DATA_BLOCK "_2015PU040U01_DB"   // DB4419
TITLE = Instance DB Unimotor:
{ S7_Optimized_Access := 'FALSE' }
AUTHOR : METIS
NAME : UNIMO_DB
VERSION : 8.0
// stored: InstanceOfName ACESYS_MOTOR
"ACESYS_MOTOR"
BEGIN
   FP_SEL.MD_OnOff := TRUE;
   FP_SEL.STW_Local := TRUE;
   FP_SEL.STW_Manual := TRUE;
   FP_SEL.STW_Single := TRUE;
   FP_SEL.Type_Unimotor := TRUE;
   FP_EN.Mode_Auto := TRUE;
   FP_EN.Mode_Man := TRUE;
   FP_EN.Mode_Loc := TRUE;
   FP_EN.Mode_SS_FP := TRUE;
   FP_SHOW.PB_Reset := TRUE;
   FP_PARM.StartWarn_Pre := 15;
   FP_PARM.RunDelay1_Pre := 5;
   FP_PARM.DelayStop_Pre := 5;
   FP_PARM.ReturnMon_Pre := 2;
   FP_PARM.AI1_Max := 19.8;
   FP_PARM.AI2_Max := 11.0;
   FP_PARM.AI3_Max := 2910.0;
   FP_PARM.AO1a_Max := 100.0;
   FP_PARM.AO2a_Max := 100.0;
   FP_PARM.AO3a_Max := 100.0;
   FP_PARM.AO1b_Max := 19.8;
   FP_PARM.AO2b_Max := 11.0;
   FP_PARM.AO3b_Max := 2910.0;
   MD := FALSE;
   SFS := FALSE;
   ES := TRUE;
   SPSET := 100.0;
   INTL.OK := TRUE;
   INTL_SEQ_STR1.OK := TRUE;
   INTL_SEQ_STR2.OK := TRUE;
   INTL_SEQ_STP.OK := TRUE;
   OK := TRUE;
   MAN := TRUE;
   CV := 100.0;
   MSW.EXT.ModeBit2 := TRUE;
   MSW.Status := 1;
   MSW.TimeStamp := 16#32F3;
   BlockInfo.Ace_Version := 80;
   BlockInfo.Ace_BuildNo := 13;
   BlockInfo.State_Act := 300;
   BlockInfo.State_Prev := 607;
   BlockInfo.DB_Number := 4419;
   FP_CMD.Manual := TRUE;
   FP_EN.PB_QStop := TRUE;
   FP_DIM.Auto := TRUE;
   FP_DIM.Local := TRUE;
   FP_DIM.Start1 := TRUE;
   FP_DIM.Start2 := TRUE;
   FP_DIM.Reset := TRUE;
   FP_SHOW.PB_Auto := TRUE;
   FP_SHOW.PB_Local := TRUE;
   FP_SHOW.PB_Manual := TRUE;
   FP_SHOW.PB_Start1 := TRUE;
   FP_SHOW.PB_Stop := TRUE;
   FP_SHOW.AI1 := TRUE;
   FP_SHOW.AI2 := TRUE;
   FP_SHOW.AI3 := TRUE;
   FP_SHOW.SP := TRUE;
   FP_SHOW.OVL := TRUE;
   FP_SHOW.SSW := TRUE;
   FP_SHOW.STALL := TRUE;
   FP_SHOW.EARTH := TRUE;
   FP_SHOW.UBAL := TRUE;
   FP_SHOW.GFA := TRUE;
   FP_SHOW.GWA := TRUE;
   FP_SHOW.BUSF := TRUE;
   FP_SHOW.DOPR := TRUE;
   FP_SHOW.DTEST := TRUE;
   FP_SHOW.LSTR1 := TRUE;
   FP_PARM.StartWarn_Acc := 15;
   FP_PARM.RunDelay1_Acc := 5;
   FP_PARM.DelayStop_Acc := 5;
   FP_PARM.ReturnMon_Acc := 2;
   FP_PARM.MD_Freq_SP := 1;
   FP_PARM.StopReason := 10;
   FP_PARM.INTL := TRUE;
   FP_PARM.INTL_SEQ_STR1 := TRUE;
   FP_PARM.INTL_SEQ_STR2 := TRUE;
   FP_PARM.INTL_SEQ_STP := TRUE;
   FP_SIM.OVL_Enable := TRUE;
   FP_SIM.RDY_Enable := TRUE;
   FP_SIM.SSW_Enable := TRUE;
   FP_SIM.TFA_Enable := TRUE;
   FP_SIM.MCC_Enable := TRUE;
   FP_SIM.DRDY_Enable := TRUE;
   FP_SIM.MD_Enable := TRUE;
   FP_SIM.GFA_Enable := TRUE;
   FP_SIM.GWA_Enable := TRUE;
   FP_SIM.STALL_Enable := TRUE;
   FP_SIM.EARTH_Enable := TRUE;
   FP_SIM.UBAL_Enable := TRUE;
   FP_SIM.BUSF_Enable := TRUE;
   FP_SIM.RET1_Enable := TRUE;
   FP_SIM.RET2_Enable := TRUE;
   FP_SIM.DOPR_Enable := TRUE;
   FP_SIM.ACK_Enable := TRUE;
   FP_SIM.LSTP_Enable := TRUE;
   FP_SIM.REM_Enable := TRUE;
   FP_SIM.SFS_Enable := TRUE;
   FP_SIM.SLS_Enable := TRUE;
   FP_SIM.ES_Enable := TRUE;
   FP_SIM.WORK.Flash_Slow := TRUE;
   AdapterBlock.Intell_Type := 282;
   AdapterBlock.VersionNo := 220;
   AdapterBlock.FuncType := 41;
   AdapterBlock.Options := 1;
   AdapterBlock.NetNo := 106;
   AdapterBlock.NodeNo := 16;
   AdapterBlock.Flash_Slow := TRUE;
   AdapterBlock.Flash_Fast := TRUE;
   AdapterBlock.MAN := TRUE;
   AdapterBlock.HMI_INT[4] := 2910;
   AdapterBlock.HMI_INT[5] := 687;
   AdapterBlock.HMI_INT[7] := 20000;
   AdapterBlock.HMI_REAL[8] := 2910.0;
   AdapterBlock.HMI_BOOL[1] := TRUE;
   AdapterBlock.HMI_BOOL[5] := TRUE;
   AdapterBlock.HMI_BOOL[6] := TRUE;
   AdapterBlock.HMI_BOOL[10] := TRUE;
   AdapterBlock.HMI_BOOL[13] := TRUE;
   AdapterBlock.HMI_BOOL[32] := TRUE;
   AdapterBlock.HMI_BOOL[34] := TRUE;
   AdapterBlock.HMI_BOOL[35] := TRUE;
   AdapterBlock.HMI_BOOL[37] := TRUE;
   AdapterBlock.HMI_BOOL[38] := TRUE;
   AdapterBlock.HMI_BOOL[39] := TRUE;
   AdapterBlock.HMI_BOOL[43] := TRUE;
   AdapterBlock.HMI_BOOL[65] := TRUE;
   AdapterBlock.HMI_BOOL[89] := TRUE;
   STATE.M_Stopped := TRUE;
   ONS.Unimotor := TRUE;
   ONS.MD_OnOff := TRUE;
   ONS.Cmd_Manual := TRUE;
   ONS.GLTP := TRUE;
   ONS.CMD_Start1 := TRUE;
   ONS.CMD_Start2 := TRUE;
   ONS.SecPulse1 := TRUE;
   StatusWork := 1;
   ModePointer := 52;
   StartWarn_Mem := 15;
   RunDelay1_Mem := 5;
   DelayStop_Mem := 5;
   ReturnMon_Mem := 2;
   ModeManual := TRUE;
   FromStateManual := TRUE;
   ChangeDir1_Done := TRUE;
   ChangeDir2_Done := TRUE;
   OUT.OK := TRUE;
   OUT.MAN := TRUE;
   OUT.INTL_OK_STAT := TRUE;
   OUT.INTL_SEQ_STR1_OK_STAT := TRUE;
   OUT.INTL_SEQ_STR2_OK_STAT := TRUE;
   OUT.INTL_SEQ_STP_OK_STAT := TRUE;
   MSW_Status_Trans := 1;
END_DATA_BLOCK

DATA_BLOCK "_2015PU041M01_DB"   // DB4420
TITLE = Instance DB Unimotor:
{ S7_Optimized_Access := 'FALSE' }
AUTHOR : METIS
NAME : UNIMO_DB
VERSION : 8.0
// stored: InstanceOfName ACESYS_MOTOR
"ACESYS_MOTOR"
BEGIN
   FP_SEL.MD_OnOff := TRUE;
   FP_SEL.STW_Local := TRUE;
   FP_SEL.STW_Manual := TRUE;
   FP_SEL.STW_Single := TRUE;
   FP_SEL.Type_Unimotor := TRUE;
   FP_EN.Mode_Auto := TRUE;
   FP_EN.Mode_Man := TRUE;
   FP_EN.Mode_Loc := TRUE;
   FP_EN.Mode_SS_FP := TRUE;
   FP_SHOW.PB_Reset := TRUE;
   FP_PARM.StartWarn_Pre := 15;
   FP_PARM.RunDelay1_Pre := 5;
   FP_PARM.DelayStop_Pre := 5;
   FP_PARM.ReturnMon_Pre := 2;
   FP_PARM.AI1_Max := 19.8;
   FP_PARM.AI2_Max := 11.0;
   FP_PARM.AI3_Max := 2910.0;
   FP_PARM.AO1a_Max := 100.0;
   FP_PARM.AO2a_Max := 100.0;
   FP_PARM.AO3a_Max := 100.0;
   FP_PARM.AO1b_Max := 19.8;
   FP_PARM.AO2b_Max := 11.0;
   FP_PARM.AO3b_Max := 2910.0;
   MD := FALSE;
   SFS := FALSE;
   ES := TRUE;
   SPSET := 100.0;
   INTL.OK := TRUE;
   INTL_SEQ_STR1.OK := TRUE;
   INTL_SEQ_STR2.OK := TRUE;
   INTL_SEQ_STP.OK := TRUE;
   OK := TRUE;
   MAN := TRUE;
   CV := 100.0;
   MSW.EXT.ModeBit2 := TRUE;
   MSW.Status := 1;
   MSW.TimeStamp := 16#32F3;
   BlockInfo.Ace_Version := 80;
   BlockInfo.Ace_BuildNo := 13;
   BlockInfo.State_Act := 300;
   BlockInfo.State_Prev := 607;
   BlockInfo.DB_Number := 4420;
   FP_CMD.Manual := TRUE;
   FP_EN.PB_QStop := TRUE;
   FP_DIM.Auto := TRUE;
   FP_DIM.Local := TRUE;
   FP_DIM.Start1 := TRUE;
   FP_DIM.Start2 := TRUE;
   FP_DIM.Reset := TRUE;
   FP_SHOW.PB_Auto := TRUE;
   FP_SHOW.PB_Local := TRUE;
   FP_SHOW.PB_Manual := TRUE;
   FP_SHOW.PB_Start1 := TRUE;
   FP_SHOW.PB_Stop := TRUE;
   FP_SHOW.AI1 := TRUE;
   FP_SHOW.AI2 := TRUE;
   FP_SHOW.AI3 := TRUE;
   FP_SHOW.SP := TRUE;
   FP_SHOW.OVL := TRUE;
   FP_SHOW.SSW := TRUE;
   FP_SHOW.STALL := TRUE;
   FP_SHOW.EARTH := TRUE;
   FP_SHOW.UBAL := TRUE;
   FP_SHOW.GFA := TRUE;
   FP_SHOW.GWA := TRUE;
   FP_SHOW.BUSF := TRUE;
   FP_SHOW.DOPR := TRUE;
   FP_SHOW.DTEST := TRUE;
   FP_SHOW.LSTR1 := TRUE;
   FP_PARM.StartWarn_Acc := 15;
   FP_PARM.RunDelay1_Acc := 5;
   FP_PARM.DelayStop_Acc := 5;
   FP_PARM.ReturnMon_Acc := 2;
   FP_PARM.MD_Freq_SP := 1;
   FP_PARM.StopReason := 11;
   FP_PARM.INTL := TRUE;
   FP_PARM.INTL_SEQ_STR1 := TRUE;
   FP_PARM.INTL_SEQ_STR2 := TRUE;
   FP_PARM.INTL_SEQ_STP := TRUE;
   FP_SIM.OVL_Enable := TRUE;
   FP_SIM.RDY_Enable := TRUE;
   FP_SIM.SSW_Enable := TRUE;
   FP_SIM.TFA_Enable := TRUE;
   FP_SIM.MCC_Enable := TRUE;
   FP_SIM.DRDY_Enable := TRUE;
   FP_SIM.MD_Enable := TRUE;
   FP_SIM.GFA_Enable := TRUE;
   FP_SIM.GWA_Enable := TRUE;
   FP_SIM.STALL_Enable := TRUE;
   FP_SIM.EARTH_Enable := TRUE;
   FP_SIM.UBAL_Enable := TRUE;
   FP_SIM.BUSF_Enable := TRUE;
   FP_SIM.RET1_Enable := TRUE;
   FP_SIM.RET2_Enable := TRUE;
   FP_SIM.DOPR_Enable := TRUE;
   FP_SIM.ACK_Enable := TRUE;
   FP_SIM.LSTP_Enable := TRUE;
   FP_SIM.REM_Enable := TRUE;
   FP_SIM.SFS_Enable := TRUE;
   FP_SIM.SLS_Enable := TRUE;
   FP_SIM.ES_Enable := TRUE;
   FP_SIM.WORK.Flash_Slow := TRUE;
   AdapterBlock.Intell_Type := 282;
   AdapterBlock.VersionNo := 220;
   AdapterBlock.FuncType := 41;
   AdapterBlock.Options := 1;
   AdapterBlock.NetNo := 106;
   AdapterBlock.NodeNo := 78;
   AdapterBlock.Flash_Slow := TRUE;
   AdapterBlock.Flash_Fast := TRUE;
   AdapterBlock.MAN := TRUE;
   AdapterBlock.HMI_INT[4] := 2910;
   AdapterBlock.HMI_INT[5] := 687;
   AdapterBlock.HMI_INT[7] := 20000;
   AdapterBlock.HMI_REAL[8] := 2910.0;
   AdapterBlock.HMI_REAL[9] := 100.0;
   AdapterBlock.HMI_REAL[10] := 100.0;
   AdapterBlock.HMI_BOOL[1] := TRUE;
   AdapterBlock.HMI_BOOL[5] := TRUE;
   AdapterBlock.HMI_BOOL[6] := TRUE;
   AdapterBlock.HMI_BOOL[10] := TRUE;
   AdapterBlock.HMI_BOOL[13] := TRUE;
   AdapterBlock.HMI_BOOL[32] := TRUE;
   AdapterBlock.HMI_BOOL[34] := TRUE;
   AdapterBlock.HMI_BOOL[35] := TRUE;
   AdapterBlock.HMI_BOOL[37] := TRUE;
   AdapterBlock.HMI_BOOL[38] := TRUE;
   AdapterBlock.HMI_BOOL[39] := TRUE;
   AdapterBlock.HMI_BOOL[43] := TRUE;
   AdapterBlock.HMI_BOOL[65] := TRUE;
   AdapterBlock.HMI_BOOL[89] := TRUE;
   STATE.M_Stopped := TRUE;
   ONS.Unimotor := TRUE;
   ONS.MD_OnOff := TRUE;
   ONS.Cmd_Manual := TRUE;
   ONS.GLTP := TRUE;
   ONS.CMD_Start1 := TRUE;
   ONS.CMD_Start2 := TRUE;
   ONS.SecPulse1 := TRUE;
   StatusWork := 1;
   ModePointer := 52;
   StartWarn_Mem := 15;
   RunDelay1_Mem := 5;
   DelayStop_Mem := 5;
   ReturnMon_Mem := 2;
   ModeManual := TRUE;
   FromStateManual := TRUE;
   ChangeDir1_Done := TRUE;
   ChangeDir2_Done := TRUE;
   OUT.OK := TRUE;
   OUT.MAN := TRUE;
   OUT.INTL_OK_STAT := TRUE;
   OUT.INTL_SEQ_STR1_OK_STAT := TRUE;
   OUT.INTL_SEQ_STR2_OK_STAT := TRUE;
   OUT.INTL_SEQ_STP_OK_STAT := TRUE;
   MSW_Status_Trans := 1;
END_DATA_BLOCK

DATA_BLOCK "_2015PU042M01_DB"   // DB4421
TITLE = Instance DB Unimotor:
{ S7_Optimized_Access := 'FALSE' }
AUTHOR : METIS
NAME : UNIMO_DB
VERSION : 8.0
// stored: InstanceOfName ACESYS_MOTOR
"ACESYS_MOTOR"
BEGIN
   FP_SEL.MD_OnOff := TRUE;
   FP_SEL.STW_Local := TRUE;
   FP_SEL.STW_Manual := TRUE;
   FP_SEL.STW_Single := TRUE;
   FP_SEL.Type_Unimotor := TRUE;
   FP_EN.Mode_Auto := TRUE;
   FP_EN.Mode_Man := TRUE;
   FP_EN.Mode_Loc := TRUE;
   FP_EN.Mode_SS_FP := TRUE;
   FP_SHOW.PB_Reset := TRUE;
   FP_PARM.StartWarn_Pre := 15;
   FP_PARM.RunDelay1_Pre := 5;
   FP_PARM.DelayStop_Pre := 5;
   FP_PARM.ReturnMon_Pre := 2;
   FP_PARM.AI1_Max := 100.0;
   FP_PARM.AI2_Max := 100.0;
   FP_PARM.AI3_Max := 100.0;
   FP_PARM.AO1a_Max := 100.0;
   FP_PARM.AO2a_Max := 100.0;
   FP_PARM.AO3a_Max := 100.0;
   FP_PARM.AO1b_Max := 100.0;
   FP_PARM.AO2b_Max := 100.0;
   FP_PARM.AO3b_Max := 100.0;
   MD := FALSE;
   SFS := FALSE;
   ES := TRUE;
   INTL.OK := TRUE;
   INTL_SEQ_STR1.OK := TRUE;
   INTL_SEQ_STR2.OK := TRUE;
   INTL_SEQ_STP.OK := TRUE;
   OK := TRUE;
   MAN := TRUE;
   MSW.EXT.ModeBit2 := TRUE;
   MSW.Status := 1;
   MSW.TimeStamp := 16#9BB1;
   BlockInfo.Ace_Version := 80;
   BlockInfo.Ace_BuildNo := 13;
   BlockInfo.State_Act := 300;
   BlockInfo.State_Prev := 607;
   BlockInfo.DB_Number := 4421;
   FP_CMD.Manual := TRUE;
   FP_EN.PB_QStop := TRUE;
   FP_DIM.Auto := TRUE;
   FP_DIM.Local := TRUE;
   FP_DIM.Start1 := TRUE;
   FP_DIM.Start2 := TRUE;
   FP_DIM.Reset := TRUE;
   FP_SHOW.PB_Auto := TRUE;
   FP_SHOW.PB_Local := TRUE;
   FP_SHOW.PB_Manual := TRUE;
   FP_SHOW.PB_Start1 := TRUE;
   FP_SHOW.PB_Stop := TRUE;
   FP_SHOW.OVL := TRUE;
   FP_SHOW.LSTP := TRUE;
   FP_SHOW.SSW := TRUE;
   FP_SHOW.DRDY := TRUE;
   FP_SHOW.STALL := TRUE;
   FP_SHOW.EARTH := TRUE;
   FP_SHOW.UBAL := TRUE;
   FP_SHOW.GFA := TRUE;
   FP_SHOW.GWA := TRUE;
   FP_SHOW.BUSF := TRUE;
   FP_SHOW.DOPR := TRUE;
   FP_SHOW.DTEST := TRUE;
   FP_SHOW.LSTR1 := TRUE;
   FP_PARM.StartWarn_Acc := 15;
   FP_PARM.RunDelay1_Acc := 5;
   FP_PARM.DelayStop_Acc := 5;
   FP_PARM.ReturnMon_Acc := 2;
   FP_PARM.MD_Freq_SP := 1;
   FP_PARM.StopReason := 99;
   FP_PARM.INTL := TRUE;
   FP_PARM.INTL_SEQ_STR1 := TRUE;
   FP_PARM.INTL_SEQ_STR2 := TRUE;
   FP_PARM.INTL_SEQ_STP := TRUE;
   FP_SIM.OVL_Enable := TRUE;
   FP_SIM.RDY_Enable := TRUE;
   FP_SIM.SSW_Enable := TRUE;
   FP_SIM.TFA_Enable := TRUE;
   FP_SIM.MCC_Enable := TRUE;
   FP_SIM.DRDY_Enable := TRUE;
   FP_SIM.MD_Enable := TRUE;
   FP_SIM.GFA_Enable := TRUE;
   FP_SIM.GWA_Enable := TRUE;
   FP_SIM.STALL_Enable := TRUE;
   FP_SIM.EARTH_Enable := TRUE;
   FP_SIM.UBAL_Enable := TRUE;
   FP_SIM.BUSF_Enable := TRUE;
   FP_SIM.RET1_Enable := TRUE;
   FP_SIM.RET2_Enable := TRUE;
   FP_SIM.DOPR_Enable := TRUE;
   FP_SIM.ACK_Enable := TRUE;
   FP_SIM.LSTP_Enable := TRUE;
   FP_SIM.REM_Enable := TRUE;
   FP_SIM.SFS_Enable := TRUE;
   FP_SIM.SLS_Enable := TRUE;
   FP_SIM.ES_Enable := TRUE;
   AdapterBlock.Intell_Type := 54;
   AdapterBlock.VersionNo := 420;
   AdapterBlock.BuildNo := 1;
   AdapterBlock.FuncType := 41;
   AdapterBlock.NetNo := 106;
   AdapterBlock.NodeNo := 64;
   AdapterBlock.MAN := TRUE;
   AdapterBlock.HMI_BOOL[4] := TRUE;
   AdapterBlock.HMI_BOOL[8] := TRUE;
   AdapterBlock.HMI_BOOL[18] := TRUE;
   AdapterBlock.HMI_BOOL[19] := TRUE;
   AdapterBlock.HMI_BOOL[20] := TRUE;
   AdapterBlock.HMI_BOOL[28] := TRUE;
   AdapterBlock.HMI_BOOL[74] := TRUE;
   STATE.M_Stopped := TRUE;
   ONS.Unimotor := TRUE;
   ONS.MD_OnOff := TRUE;
   ONS.Cmd_Manual := TRUE;
   ONS.GLTP := TRUE;
   ONS.CMD_Start1 := TRUE;
   ONS.CMD_Start2 := TRUE;
   ONS.SecPulse1 := TRUE;
   StatusWork := 1;
   ModePointer := 52;
   StartWarn_Mem := 15;
   RunDelay1_Mem := 5;
   DelayStop_Mem := 5;
   ReturnMon_Mem := 2;
   ModeManual := TRUE;
   FromStateManual := TRUE;
   ChangeDir1_Done := TRUE;
   ChangeDir2_Done := TRUE;
   OUT.OK := TRUE;
   OUT.MAN := TRUE;
   OUT.INTL_OK_STAT := TRUE;
   OUT.INTL_SEQ_STR1_OK_STAT := TRUE;
   OUT.INTL_SEQ_STR2_OK_STAT := TRUE;
   OUT.INTL_SEQ_STP_OK_STAT := TRUE;
   MSW_Status_Trans := 1;
END_DATA_BLOCK

DATA_BLOCK "_MTR_SPARE_DB"   // DB4422
TITLE = Instance DB Unimotor:
{ S7_Optimized_Access := 'FALSE' }
AUTHOR : METIS
NAME : UNIMO_DB
VERSION : 8.0
// stored: InstanceOfName ACESYS_MOTOR
"ACESYS_MOTOR"
BEGIN
   FP_SEL.MD_OnOff := TRUE;
   FP_SEL.STW_Local := TRUE;
   FP_SEL.STW_Manual := TRUE;
   FP_SEL.STW_Single := TRUE;
   FP_SEL.Type_Unimotor := TRUE;
   FP_EN.Mode_Auto := TRUE;
   FP_EN.Mode_Man := TRUE;
   FP_EN.Mode_Loc := TRUE;
   FP_EN.Mode_SS_FP := TRUE;
   FP_SHOW.PB_Reset := TRUE;
   FP_PARM.StartWarn_Pre := 15;
   FP_PARM.RunDelay1_Pre := 5;
   FP_PARM.DelayStop_Pre := 5;
   FP_PARM.ReturnMon_Pre := 2;
   FP_PARM.AI1_Max := 100.0;
   FP_PARM.AI2_Max := 100.0;
   FP_PARM.AI3_Max := 100.0;
   FP_PARM.AO1a_Max := 100.0;
   FP_PARM.AO2a_Max := 100.0;
   FP_PARM.AO3a_Max := 100.0;
   FP_PARM.AO1b_Max := 100.0;
   FP_PARM.AO2b_Max := 100.0;
   FP_PARM.AO3b_Max := 100.0;
   MD := FALSE;
   SFS := FALSE;
   ES := TRUE;
   INTL.OK := TRUE;
   INTL_SEQ_STR1.OK := TRUE;
   INTL_SEQ_STR2.OK := TRUE;
   INTL_SEQ_STP.OK := TRUE;
   OK := TRUE;
   MAN := TRUE;
   MSW.EXT.ModeBit2 := TRUE;
   MSW.Status := 1;
   MSW.TimeStamp := 16#9BB1;
   BlockInfo.Ace_Version := 80;
   BlockInfo.Ace_BuildNo := 13;
   BlockInfo.State_Act := 300;
   BlockInfo.State_Prev := 607;
   BlockInfo.DB_Number := 4421;
   FP_CMD.Manual := TRUE;
   FP_EN.PB_QStop := TRUE;
   FP_DIM.Auto := TRUE;
   FP_DIM.Local := TRUE;
   FP_DIM.Start1 := TRUE;
   FP_DIM.Start2 := TRUE;
   FP_DIM.Reset := TRUE;
   FP_SHOW.PB_Auto := TRUE;
   FP_SHOW.PB_Local := TRUE;
   FP_SHOW.PB_Manual := TRUE;
   FP_SHOW.PB_Start1 := TRUE;
   FP_SHOW.PB_Stop := TRUE;
   FP_SHOW.OVL := TRUE;
   FP_SHOW.LSTP := TRUE;
   FP_SHOW.SSW := TRUE;
   FP_SHOW.DRDY := TRUE;
   FP_SHOW.STALL := TRUE;
   FP_SHOW.EARTH := TRUE;
   FP_SHOW.UBAL := TRUE;
   FP_SHOW.GFA := TRUE;
   FP_SHOW.GWA := TRUE;
   FP_SHOW.BUSF := TRUE;
   FP_SHOW.DOPR := TRUE;
   FP_SHOW.DTEST := TRUE;
   FP_SHOW.LSTR1 := TRUE;
   FP_PARM.StartWarn_Acc := 15;
   FP_PARM.RunDelay1_Acc := 5;
   FP_PARM.DelayStop_Acc := 5;
   FP_PARM.ReturnMon_Acc := 2;
   FP_PARM.MD_Freq_SP := 1;
   FP_PARM.StopReason := 99;
   FP_PARM.INTL := TRUE;
   FP_PARM.INTL_SEQ_STR1 := TRUE;
   FP_PARM.INTL_SEQ_STR2 := TRUE;
   FP_PARM.INTL_SEQ_STP := TRUE;
   FP_SIM.OVL_Enable := TRUE;
   FP_SIM.RDY_Enable := TRUE;
   FP_SIM.SSW_Enable := TRUE;
   FP_SIM.TFA_Enable := TRUE;
   FP_SIM.MCC_Enable := TRUE;
   FP_SIM.DRDY_Enable := TRUE;
   FP_SIM.MD_Enable := TRUE;
   FP_SIM.GFA_Enable := TRUE;
   FP_SIM.GWA_Enable := TRUE;
   FP_SIM.STALL_Enable := TRUE;
   FP_SIM.EARTH_Enable := TRUE;
   FP_SIM.UBAL_Enable := TRUE;
   FP_SIM.BUSF_Enable := TRUE;
   FP_SIM.RET1_Enable := TRUE;
   FP_SIM.RET2_Enable := TRUE;
   FP_SIM.DOPR_Enable := TRUE;
   FP_SIM.ACK_Enable := TRUE;
   FP_SIM.LSTP_Enable := TRUE;
   FP_SIM.REM_Enable := TRUE;
   FP_SIM.SFS_Enable := TRUE;
   FP_SIM.SLS_Enable := TRUE;
   FP_SIM.ES_Enable := TRUE;
   AdapterBlock.Intell_Type := 54;
   AdapterBlock.VersionNo := 420;
   AdapterBlock.BuildNo := 1;
   AdapterBlock.FuncType := 41;
   AdapterBlock.NetNo := 106;
   AdapterBlock.NodeNo := 64;
   AdapterBlock.MAN := TRUE;
   AdapterBlock.HMI_BOOL[4] := TRUE;
   AdapterBlock.HMI_BOOL[8] := TRUE;
   AdapterBlock.HMI_BOOL[18] := TRUE;
   AdapterBlock.HMI_BOOL[19] := TRUE;
   AdapterBlock.HMI_BOOL[20] := TRUE;
   AdapterBlock.HMI_BOOL[28] := TRUE;
   AdapterBlock.HMI_BOOL[74] := TRUE;
   STATE.M_Stopped := TRUE;
   ONS.Unimotor := TRUE;
   ONS.MD_OnOff := TRUE;
   ONS.Cmd_Manual := TRUE;
   ONS.GLTP := TRUE;
   ONS.CMD_Start1 := TRUE;
   ONS.CMD_Start2 := TRUE;
   ONS.SecPulse1 := TRUE;
   StatusWork := 1;
   ModePointer := 52;
   StartWarn_Mem := 15;
   RunDelay1_Mem := 5;
   DelayStop_Mem := 5;
   ReturnMon_Mem := 2;
   ModeManual := TRUE;
   FromStateManual := TRUE;
   ChangeDir1_Done := TRUE;
   ChangeDir2_Done := TRUE;
   OUT.OK := TRUE;
   OUT.MAN := TRUE;
   OUT.INTL_OK_STAT := TRUE;
   OUT.INTL_SEQ_STR1_OK_STAT := TRUE;
   OUT.INTL_SEQ_STR2_OK_STAT := TRUE;
   OUT.INTL_SEQ_STP_OK_STAT := TRUE;
   MSW_Status_Trans := 1;
END_DATA_BLOCK

DATA_BLOCK "_2015PU035U01_DB"   // DB4433
TITLE = Instance DB Unimotor:
{ S7_Optimized_Access := 'FALSE' }
AUTHOR : METIS
NAME : UNIMO_DB
VERSION : 8.0
// stored: InstanceOfName ACESYS_MOTOR
"ACESYS_MOTOR"
BEGIN
   FP_SEL.MD_OnOff := TRUE;
   FP_SEL.STW_Local := TRUE;
   FP_SEL.STW_Manual := TRUE;
   FP_SEL.STW_Single := TRUE;
   FP_SEL.Type_Unimotor := TRUE;
   FP_EN.Mode_Auto := TRUE;
   FP_EN.Mode_Man := TRUE;
   FP_EN.Mode_Loc := TRUE;
   FP_EN.Mode_SS_FP := TRUE;
   FP_SHOW.PB_Reset := TRUE;
   FP_PARM.StartWarn_Pre := 15;
   FP_PARM.RunDelay1_Pre := 5;
   FP_PARM.DelayStop_Pre := 5;
   FP_PARM.ReturnMon_Pre := 2;
   FP_PARM.AI1_Max := 100.0;
   FP_PARM.AI2_Max := 100.0;
   FP_PARM.AI3_Max := 100.0;
   FP_PARM.AO1a_Max := 100.0;
   FP_PARM.AO2a_Max := 100.0;
   FP_PARM.AO3a_Max := 100.0;
   FP_PARM.AO1b_Max := 100.0;
   FP_PARM.AO2b_Max := 100.0;
   FP_PARM.AO3b_Max := 100.0;
   MD := FALSE;
   SFS := FALSE;
   SLS := TRUE;
   ES := TRUE;
   SPSET := 20.0;
   INTL.OK := TRUE;
   INTL_SEQ_STR1.OK := TRUE;
   INTL_SEQ_STR2.OK := TRUE;
   INTL_SEQ_STP.OK := TRUE;
   OK := TRUE;
   MAN := TRUE;
   CV := 20.0;
   MSW.EXT.ModeBit2 := TRUE;
   MSW.Status := 1;
   MSW.TimeStamp := 16#A9DD;
   BlockInfo.Ace_Version := 80;
   BlockInfo.Ace_BuildNo := 13;
   BlockInfo.State_Act := 300;
   BlockInfo.State_Prev := 305;
   BlockInfo.DB_Number := 4433;
   FP_CMD.Manual := TRUE;
   FP_EN.PB_QStop := TRUE;
   FP_DIM.Auto := TRUE;
   FP_DIM.Local := TRUE;
   FP_DIM.Start1 := TRUE;
   FP_DIM.Start2 := TRUE;
   FP_DIM.Reset := TRUE;
   FP_SHOW.PB_Auto := TRUE;
   FP_SHOW.PB_Local := TRUE;
   FP_SHOW.PB_Manual := TRUE;
   FP_SHOW.PB_Start1 := TRUE;
   FP_SHOW.PB_Stop := TRUE;
   FP_SHOW.AI1 := TRUE;
   FP_SHOW.AI2 := TRUE;
   FP_SHOW.AI3 := TRUE;
   FP_SHOW.SP := TRUE;
   FP_SHOW.OVL := TRUE;
   FP_SHOW.SSW := TRUE;
   FP_SHOW.STALL := TRUE;
   FP_SHOW.EARTH := TRUE;
   FP_SHOW.UBAL := TRUE;
   FP_SHOW.GFA := TRUE;
   FP_SHOW.GWA := TRUE;
   FP_SHOW.BUSF := TRUE;
   FP_SHOW.DOPR := TRUE;
   FP_SHOW.DTEST := TRUE;
   FP_SHOW.LSTR1 := TRUE;
   FP_PARM.StartWarn_Acc := 15;
   FP_PARM.RunDelay1_Acc := 5;
   FP_PARM.DelayStop_Acc := 5;
   FP_PARM.ReturnMon_Acc := 2;
   FP_PARM.MD_Freq_SP := 1;
   FP_PARM.StopReason := 3;
   FP_PARM.INTL := TRUE;
   FP_PARM.INTL_SEQ_STR1 := TRUE;
   FP_PARM.INTL_SEQ_STR2 := TRUE;
   FP_PARM.INTL_SEQ_STP := TRUE;
   FP_SIM.OVL_Enable := TRUE;
   FP_SIM.RDY_Enable := TRUE;
   FP_SIM.SSW_Enable := TRUE;
   FP_SIM.TFA_Enable := TRUE;
   FP_SIM.MCC_Enable := TRUE;
   FP_SIM.DRDY_Enable := TRUE;
   FP_SIM.MD_Enable := TRUE;
   FP_SIM.GFA_Enable := TRUE;
   FP_SIM.GWA_Enable := TRUE;
   FP_SIM.STALL_Enable := TRUE;
   FP_SIM.EARTH_Enable := TRUE;
   FP_SIM.UBAL_Enable := TRUE;
   FP_SIM.BUSF_Enable := TRUE;
   FP_SIM.RET1_Enable := TRUE;
   FP_SIM.RET2_Enable := TRUE;
   FP_SIM.DOPR_Enable := TRUE;
   FP_SIM.ACK_Enable := TRUE;
   FP_SIM.LSTP_Enable := TRUE;
   FP_SIM.REM_Enable := TRUE;
   FP_SIM.SFS_Enable := TRUE;
   FP_SIM.SLS_Enable := TRUE;
   FP_SIM.ES_Enable := TRUE;
   AdapterBlock.Intell_Type := 282;
   AdapterBlock.VersionNo := 220;
   AdapterBlock.FuncType := 41;
   AdapterBlock.Options := 1;
   AdapterBlock.NetNo := 106;
   AdapterBlock.NodeNo := 75;
   AdapterBlock.MAN := TRUE;
   AdapterBlock.HMI_INT[7] := 1000;
   AdapterBlock.HMI_INT[9] := 3;
   AdapterBlock.HMI_INT[10] := 2;
   AdapterBlock.HMI_INT[11] := 6;
   AdapterBlock.HMI_REAL[9] := 100.0;
   AdapterBlock.HMI_REAL[10] := 100.0;
   AdapterBlock.HMI_REAL[12] := 100.0;
   AdapterBlock.HMI_BOOL[1] := TRUE;
   AdapterBlock.HMI_BOOL[2] := TRUE;
   AdapterBlock.HMI_BOOL[9] := TRUE;
   AdapterBlock.HMI_BOOL[15] := TRUE;
   AdapterBlock.HMI_BOOL[17] := TRUE;
   AdapterBlock.HMI_BOOL[18] := TRUE;
   AdapterBlock.HMI_BOOL[34] := TRUE;
   AdapterBlock.HMI_BOOL[35] := TRUE;
   AdapterBlock.HMI_BOOL[65] := TRUE;
   AdapterBlock.HMI_BOOL[89] := TRUE;
   STATE.M_Stopped := TRUE;
   ONS.Unimotor := TRUE;
   ONS.MD_OnOff := TRUE;
   ONS.Cmd_Manual := TRUE;
   ONS.GLTP := TRUE;
   ONS.CMD_Start1 := TRUE;
   ONS.CMD_Start2 := TRUE;
   ONS.SecPulse1 := TRUE;
   StatusWork := 1;
   ModePointer := 52;
   StartWarn_Mem := 15;
   RunDelay1_Mem := 5;
   DelayStop_Mem := 5;
   ReturnMon_Mem := 2;
   ModeManual := TRUE;
   FromStateManual := TRUE;
   ChangeDir1_Done := TRUE;
   ChangeDir2_Done := TRUE;
   OUT.OK := TRUE;
   OUT.MAN := TRUE;
   OUT.INTL_OK_STAT := TRUE;
   OUT.INTL_SEQ_STR1_OK_STAT := TRUE;
   OUT.INTL_SEQ_STR2_OK_STAT := TRUE;
   OUT.INTL_SEQ_STP_OK_STAT := TRUE;
   MSW_Status_Trans := 1;
END_DATA_BLOCK

DATA_BLOCK "_2015PU027Y01_DB"   // DB4434
{ S7_Optimized_Access := 'FALSE' }
AUTHOR : FLSmidth
FAMILY : ACESYS
NAME : VALVE
VERSION : 8.0
// stored: InstanceOfName ACESYS_VALVE
"ACESYS_VALVE"
BEGIN
END_DATA_BLOCK

DATA_BLOCK "_2015PU028Y01_DB"   // DB4435
{ S7_Optimized_Access := 'FALSE' }
AUTHOR : FLSmidth
FAMILY : ACESYS
NAME : VALVE
VERSION : 8.0
// stored: InstanceOfName ACESYS_VALVE
"ACESYS_VALVE"
BEGIN
END_DATA_BLOCK

DATA_BLOCK "_2010CV300N01T01_DB"   // DB5000
TITLE = Instance DB Analog:
{ S7_Optimized_Access := 'FALSE' }
AUTHOR : METIS
NAME : ANA_DB
VERSION : 8.0
// stored: InstanceOfName ACESYS_ANALOG
"ACESYS_ANALOG"
BEGIN
   FP_EN.ParentSupress := TRUE;
   FP_EN.ParentSupressUnit := TRUE;
   FP_EN.Hysteresis := TRUE;
   FP_PARM.Scale_Max := 200.0;
   FP_PARM.Grad_Pos := 0.0;
   FP_PARM.Grad_Neg := 0.0;
   FP_PARM.OpenLoopDelay_Pre := 2;
   FP_PARM.Gradient_Time_Pre := 10;
   FP_PARM.Alarm_Hyst := 1.0;
   FP_PARM.OverRangeDelay_Pre := 2;
   FP_SIM.Value_Enable := TRUE;
   FP_SIM.Gain := 1.0;
   IN := 41.90176;
   U_RANGE := TRUE;
   O_RANGE := TRUE;
   SIG_FAULT := TRUE;
   EnConfig := TRUE;
   AEN := TRUE;
   PV_NORM := 41.90176;
   PV_SCAL := 54.75442;
   AL_H3 := TRUE;
   AL_H2 := TRUE;
   AL_H1 := TRUE;
   AL_L1 := TRUE;
   AL_L2 := TRUE;
   AL_L3 := TRUE;
   SIG_OK := TRUE;
   LIM_H2 := TRUE;
   LIM_H1 := TRUE;
   MSW.VALUE := 54.75442;
   MSW.TRIGVALUE := -53.03819;
   MSW.EXT.AlarmWarnUnAck := TRUE;
   MSW.EXT.Operation := TRUE;
   MSW.Status := 1;
   MSW.TimeStamp := 16#97DF;
   BlockInfo.Ace_Version := 80;
   BlockInfo.Ace_BuildNo := 3;
   BlockInfo.DB_Number := 5000;
   FP_EN.Alarm_H2 := TRUE;
   FP_EN.Alarm_H1 := TRUE;
   FP_EN.AlarmDelay_H2 := TRUE;
   FP_EN.AlarmDelay_H1 := TRUE;
   FP_PARM.Scale_Min := -50.0;
   FP_PARM.Gradient_Time_ACC := 10;
   FP_PARM.AlarmLimit_H2 := 85.0;
   FP_PARM.AlarmLimit_H1 := 80.0;
   FP_PARM.AlarmDelay_H2_Pre := 2;
   FP_PARM.AlarmDelay_H2_Acc := 2;
   FP_PARM.AlarmDelay_H1_Pre := 2;
   FP_PARM.AlarmDelay_H1_Acc := 2;
   FP_PARM.OpenLoopDelay_Acc := 2;
   FP_PARM.OverRangeDelay_Acc := 2;
   ONS.SecPulse1 := TRUE;
   FIBUS_SubStatus := 16#FF;
   FIBUS_Quality := 16#FF;
   FIBUS_Limit := 16#FF;
   Result_Smooth := 41.90176;
   DampXEA := 41.90176;
   StatusWork := 1;
   AlarmDelay_H2_Mem := 2;
   AlarmDelay_H1_Mem := 2;
   GradientTime_Mem := 10;
   AlarmDelay_OpenLoop_Mem := 2;
   AlarmDelay_OverRange_Mem := 2;
   ScaledValue := 54.75442;
   Grad_OldValue := 54.75442;
   HystCalc := 2.5;
   OUT.PV_NORM := 41.90176;
   OUT.PV_SCAL := 54.75442;
   OUT.AL_H3 := TRUE;
   OUT.AL_H2 := TRUE;
   OUT.AL_H1 := TRUE;
   OUT.AL_L1 := TRUE;
   OUT.AL_L2 := TRUE;
   OUT.AL_L3 := TRUE;
   OUT.SIG_OK := TRUE;
   OUT.LIM_H2 := TRUE;
   OUT.LIM_H1 := TRUE;
   MSW_Status_Trans := 1;
END_DATA_BLOCK

DATA_BLOCK "_2010CV300U01I01_DB"   // DB5001
TITLE = Instance DB Analog:
{ S7_Optimized_Access := 'FALSE' }
AUTHOR : METIS
NAME : ANA_DB
VERSION : 8.0
// stored: InstanceOfName ACESYS_ANALOG
"ACESYS_ANALOG"
BEGIN
   FP_EN.Hysteresis := TRUE;
   FP_PARM.Scale_Max := 487.0;
   FP_PARM.Grad_Pos := 0.0;
   FP_PARM.Grad_Neg := 0.0;
   FP_PARM.OpenLoopDelay_Pre := 2;
   FP_PARM.Gradient_Time_Pre := 10;
   FP_PARM.Alarm_Hyst := 1.0;
   FP_PARM.OverRangeDelay_Pre := 2;
   FP_SIM.Value_Enable := TRUE;
   FP_SIM.Gain := 1.0;
   SIG_TYPE := 1;
   IN := 251.3;
   U_RANGE := TRUE;
   O_RANGE := TRUE;
   SIG_FAULT := TRUE;
   EnConfig := TRUE;
   AEN := TRUE;
   PV_NORM := 51.60164;
   PV_SCAL := 251.3;
   AL_H3 := TRUE;
   AL_H2 := TRUE;
   AL_H1 := TRUE;
   AL_L1 := TRUE;
   AL_L2 := TRUE;
   AL_L3 := TRUE;
   SIG_OK := TRUE;
   LIM_H2 := TRUE;
   LIM_H1 := TRUE;
   MSW.VALUE := 251.3;
   MSW.TRIGVALUE := 294.1;
   MSW.EXT.AlarmWarnUnAck := TRUE;
   MSW.EXT.Operation := TRUE;
   MSW.Status := 1;
   MSW.TimeStamp := 16#ADFA;
   BlockInfo.Ace_Version := 80;
   BlockInfo.Ace_BuildNo := 3;
   BlockInfo.DB_Number := 5001;
   FP_EN.Alarm_H3 := TRUE;
   FP_EN.Alarm_H2 := TRUE;
   FP_EN.Alarm_H1 := TRUE;
   FP_EN.AlarmDelay_H3 := TRUE;
   FP_EN.AlarmDelay_H2 := TRUE;
   FP_EN.U_Range_Warn := FALSE;
   FP_EN.O_Range_Warn := FALSE;
   FP_PARM.Gradient_Time_ACC := 10;
   FP_PARM.AlarmLimit_H3 := 350.0;
   FP_PARM.AlarmLimit_H2 := 320.0;
   FP_PARM.AlarmLimit_H1 := 300.0;
   FP_PARM.AlarmDelay_H3_Pre := 30;
   FP_PARM.AlarmDelay_H3_Acc := 30;
   FP_PARM.AlarmDelay_H2_Pre := 1;
   FP_PARM.AlarmDelay_H2_Acc := 1;
   FP_PARM.OpenLoopDelay_Acc := 2;
   FP_PARM.OverRangeDelay_Acc := 2;
   ONS.SecPulse1 := TRUE;
   FIBUS_SubStatus := 16#FF;
   FIBUS_Quality := 16#FF;
   FIBUS_Limit := 16#FF;
   Result_Smooth := 51.60164;
   DampXEA := 51.60164;
   StatusWork := 1;
   AlarmDelay_H3_Mem := 30;
   AlarmDelay_H2_Mem := 1;
   GradientTime_Mem := 10;
   AlarmDelay_OpenLoop_Mem := 2;
   AlarmDelay_OverRange_Mem := 2;
   ScaledValue := 251.3;
   Grad_OldValue := 251.3;
   HystCalc := 4.87;
   OUT.PV_NORM := 51.60164;
   OUT.PV_SCAL := 251.3;
   OUT.AL_H3 := TRUE;
   OUT.AL_H2 := TRUE;
   OUT.AL_H1 := TRUE;
   OUT.AL_L1 := TRUE;
   OUT.AL_L2 := TRUE;
   OUT.AL_L3 := TRUE;
   OUT.SIG_OK := TRUE;
   OUT.LIM_H2 := TRUE;
   OUT.LIM_H1 := TRUE;
   MSW_Status_Trans := 1;
END_DATA_BLOCK

DATA_BLOCK "_2010CV300U01J01_DB"   // DB5002
TITLE = Instance DB Analog:
{ S7_Optimized_Access := 'FALSE' }
AUTHOR : METIS
NAME : ANA_DB
VERSION : 8.0
// stored: InstanceOfName ACESYS_ANALOG
"ACESYS_ANALOG"
BEGIN
   FP_EN.ParentSupress := TRUE;
   FP_EN.ParentSupressUnit := TRUE;
   FP_EN.Hysteresis := TRUE;
   FP_PARM.OverRangeDelay_Pre := 2;
   FP_PARM.Grad_Pos := 0.0;
   FP_PARM.Grad_Neg := 0.0;
   FP_PARM.OpenLoopDelay_Pre := 2;
   FP_PARM.Gradient_Time_Pre := 10;
   FP_PARM.Alarm_Hyst := 1.0;
   FP_SIM.Value_Enable := TRUE;
   FP_SIM.Gain := 1.0;
   SIG_TYPE := 1;
   IN := 140.0;
   U_RANGE := TRUE;
   O_RANGE := TRUE;
   SIG_FAULT := TRUE;
   EnConfig := TRUE;
   AEN := TRUE;
   PV_NORM := 140.0;
   PV_SCAL := 140.0;
   AL_H3 := TRUE;
   AL_H2 := TRUE;
   AL_H1 := TRUE;
   AL_L1 := TRUE;
   AL_L2 := TRUE;
   AL_L3 := TRUE;
   SIG_OK := TRUE;
   LIM_H2 := TRUE;
   LIM_H1 := TRUE;
   MSW.VALUE := 140.0;
   MSW.EXT.AlarmWarnUnAck := TRUE;
   MSW.EXT.Operation := TRUE;
   MSW.Status := 1;
   MSW.TimeStamp := 16#3928;
   BlockInfo.Ace_Version := 80;
   BlockInfo.Ace_BuildNo := 3;
   BlockInfo.DB_Number := 5002;
   FP_EN.U_Range_Warn := FALSE;
   FP_EN.O_Range_Warn := FALSE;
   FP_PARM.Gradient_Time_ACC := 10;
   FP_PARM.OpenLoopDelay_Acc := 2;
   FP_PARM.OverRangeDelay_Acc := 2;
   ONS.SecPulse1 := TRUE;
   FIBUS_SubStatus := 16#FF;
   FIBUS_Quality := 16#FF;
   FIBUS_Limit := 16#FF;
   Result_Smooth := 140.0;
   DampXEA := 140.0;
   StatusWork := 1;
   GradientTime_Mem := 10;
   AlarmDelay_OpenLoop_Mem := 2;
   AlarmDelay_OverRange_Mem := 2;
   ScaledValue := 140.0;
   Grad_OldValue := 140.0;
   HystCalc := 1.0;
   OUT.PV_NORM := 140.0;
   OUT.PV_SCAL := 140.0;
   OUT.AL_H3 := TRUE;
   OUT.AL_H2 := TRUE;
   OUT.AL_H1 := TRUE;
   OUT.AL_L1 := TRUE;
   OUT.AL_L2 := TRUE;
   OUT.AL_L3 := TRUE;
   OUT.SIG_OK := TRUE;
   OUT.LIM_H2 := TRUE;
   OUT.LIM_H1 := TRUE;
   MSW_Status_Trans := 1;
END_DATA_BLOCK

DATA_BLOCK "_2010CV300U01S01_DB"   // DB5003
TITLE = Instance DB Analog:
{ S7_Optimized_Access := 'FALSE' }
AUTHOR : METIS
NAME : ANA_DB
VERSION : 8.0
// stored: InstanceOfName ACESYS_ANALOG
"ACESYS_ANALOG"
BEGIN
   FP_EN.ParentSupress := TRUE;
   FP_EN.ParentSupressUnit := TRUE;
   FP_EN.Hysteresis := TRUE;
   FP_PARM.Grad_Pos := 0.0;
   FP_PARM.Grad_Neg := 0.0;
   FP_PARM.OpenLoopDelay_Pre := 2;
   FP_PARM.Gradient_Time_Pre := 10;
   FP_PARM.Alarm_Hyst := 1.0;
   FP_PARM.OverRangeDelay_Pre := 2;
   FP_SIM.Value_Enable := TRUE;
   FP_SIM.Gain := 1.0;
   IN := 110.9;
   U_RANGE := TRUE;
   O_RANGE := TRUE;
   SIG_FAULT := TRUE;
   EnConfig := TRUE;
   AEN := TRUE;
   PV_NORM := 110.9;
   PV_SCAL := 110.9;
   AL_H3 := TRUE;
   AL_H2 := TRUE;
   AL_H1 := TRUE;
   AL_L1 := TRUE;
   AL_L2 := TRUE;
   AL_L3 := TRUE;
   SIG_OK := TRUE;
   LIM_H2 := TRUE;
   LIM_H1 := TRUE;
   MSW.VALUE := 110.9;
   MSW.EXT.AlarmWarnUnAck := TRUE;
   MSW.EXT.Operation := TRUE;
   MSW.Status := 1;
   MSW.TimeStamp := 16#3928;
   BlockInfo.Ace_Version := 80;
   BlockInfo.Ace_BuildNo := 3;
   BlockInfo.DB_Number := 5003;
   FP_EN.U_Range_Warn := FALSE;
   FP_EN.O_Range_Warn := FALSE;
   FP_PARM.Gradient_Time_ACC := 10;
   FP_PARM.OpenLoopDelay_Acc := 2;
   FP_PARM.OverRangeDelay_Acc := 2;
   ONS.SecPulse1 := TRUE;
   FIBUS_SubStatus := 16#FF;
   FIBUS_Quality := 16#FF;
   FIBUS_Limit := 16#FF;
   Result_Smooth := 110.9;
   DampXEA := 110.9;
   StatusWork := 1;
   GradientTime_Mem := 10;
   AlarmDelay_OpenLoop_Mem := 2;
   AlarmDelay_OverRange_Mem := 2;
   ScaledValue := 110.9;
   Grad_OldValue := 110.9;
   HystCalc := 1.0;
   OUT.PV_NORM := 110.9;
   OUT.PV_SCAL := 110.9;
   OUT.AL_H3 := TRUE;
   OUT.AL_H2 := TRUE;
   OUT.AL_H1 := TRUE;
   OUT.AL_L1 := TRUE;
   OUT.AL_L2 := TRUE;
   OUT.AL_L3 := TRUE;
   OUT.SIG_OK := TRUE;
   OUT.LIM_H2 := TRUE;
   OUT.LIM_H1 := TRUE;
   MSW_Status_Trans := 1;
END_DATA_BLOCK

DATA_BLOCK "_2010CV180U01I01_DB"   // DB5004
TITLE = Instance DB Analog: _2010CV180U01I01
{ S7_Optimized_Access := 'FALSE' }
AUTHOR : METIS
NAME : ANA_DB
VERSION : 8.0
// stored: InstanceOfName ACESYS_ANALOG
"ACESYS_ANALOG"
BEGIN
   FP_EN.Hysteresis := TRUE;
   FP_PARM.Grad_Pos := 0.0;
   FP_PARM.Grad_Neg := 0.0;
   FP_PARM.OpenLoopDelay_Pre := 2;
   FP_PARM.Gradient_Time_Pre := 10;
   FP_PARM.Alarm_Hyst := 1.0;
   FP_PARM.OverRangeDelay_Pre := 2;
   FP_SIM.Value_Enable := TRUE;
   FP_SIM.Gain := 1.0;
   SIG_TYPE := 1;
   IN := 9.15;
   U_RANGE := TRUE;
   O_RANGE := TRUE;
   SIG_FAULT := TRUE;
   EnConfig := TRUE;
   AEN := TRUE;
   PV_NORM := 9.15;
   PV_SCAL := 9.15;
   AL_H3 := TRUE;
   AL_H2 := TRUE;
   AL_H1 := TRUE;
   AL_L1 := TRUE;
   AL_L2 := TRUE;
   AL_L3 := TRUE;
   SIG_OK := TRUE;
   LIM_H2 := TRUE;
   MSW.VALUE := 9.15;
   MSW.TRIGVALUE := 6.9;
   MSW.EXT.AlarmWarnUnAck := TRUE;
   MSW.EXT.Operation := TRUE;
   MSW.Status := 1;
   MSW.TimeStamp := 16#3705;
   BlockInfo.Ace_Version := 80;
   BlockInfo.Ace_BuildNo := 3;
   BlockInfo.DB_Number := 5004;
   FP_EN.Alarm_H3 := TRUE;
   FP_EN.Alarm_H2 := TRUE;
   FP_EN.Alarm_H1 := TRUE;
   FP_EN.AlarmDelay_H3 := TRUE;
   FP_EN.AlarmDelay_H2 := TRUE;
   FP_EN.U_Range_Warn := FALSE;
   FP_EN.O_Range_Warn := FALSE;
   FP_PARM.Gradient_Time_ACC := 10;
   FP_PARM.AlarmLimit_H3 := 100.0;
   FP_PARM.AlarmLimit_H2 := 90.0;
   FP_PARM.AlarmLimit_H1 := 70.0;
   FP_PARM.AlarmDelay_H3_Pre := 10;
   FP_PARM.AlarmDelay_H3_Acc := 10;
   FP_PARM.AlarmDelay_H2_Pre := 5;
   FP_PARM.AlarmDelay_H2_Acc := 5;
   FP_PARM.OpenLoopDelay_Acc := 2;
   FP_PARM.OverRangeDelay_Acc := 2;
   FP_PARM.AuxLimit_H1_Value := 55.0;
   ONS.SecPulse1 := TRUE;
   FIBUS_SubStatus := 16#FF;
   FIBUS_Quality := 16#FF;
   FIBUS_Limit := 16#FF;
   Result_Smooth := 9.15;
   DampXEA := 9.15;
   StatusWork := 1;
   AlarmDelay_H3_Mem := 10;
   AlarmDelay_H2_Mem := 5;
   GradientTime_Mem := 10;
   AlarmDelay_OpenLoop_Mem := 2;
   AlarmDelay_OverRange_Mem := 2;
   ScaledValue := 9.15;
   Grad_OldValue := 9.15;
   HystCalc := 1.0;
   OUT.PV_NORM := 9.15;
   OUT.PV_SCAL := 9.15;
   OUT.AL_H3 := TRUE;
   OUT.AL_H2 := TRUE;
   OUT.AL_H1 := TRUE;
   OUT.AL_L1 := TRUE;
   OUT.AL_L2 := TRUE;
   OUT.AL_L3 := TRUE;
   OUT.SIG_OK := TRUE;
   OUT.LIM_H2 := TRUE;
   MSW_Status_Trans := 1;
END_DATA_BLOCK

DATA_BLOCK "_2010CV180U01J01_DB"   // DB5005
{ S7_Optimized_Access := 'FALSE' }
AUTHOR : FLSmidth
FAMILY : ACESYS
NAME : ANALOG
VERSION : 8.0
// stored: InstanceOfName ACESYS_ANALOG
"ACESYS_ANALOG"
BEGIN
END_DATA_BLOCK

DATA_BLOCK "_2010CV180U01S01_DB"   // DB5006
TITLE = Instance DB Analog: _2010CV180U01S01
{ S7_Optimized_Access := 'FALSE' }
AUTHOR : METIS
NAME : ANA_DB
VERSION : 8.0
// stored: InstanceOfName ACESYS_ANALOG
"ACESYS_ANALOG"
BEGIN
   FP_EN.ParentSupress := TRUE;
   FP_EN.ParentSupressUnit := TRUE;
   FP_EN.Hysteresis := TRUE;
   FP_PARM.Grad_Pos := 0.0;
   FP_PARM.Grad_Neg := 0.0;
   FP_PARM.OpenLoopDelay_Pre := 2;
   FP_PARM.Gradient_Time_Pre := 10;
   FP_PARM.Alarm_Hyst := 1.0;
   FP_PARM.OverRangeDelay_Pre := 2;
   FP_SIM.Value_Enable := TRUE;
   FP_SIM.Gain := 1.0;
   IN := 90.0;
   U_RANGE := TRUE;
   O_RANGE := TRUE;
   SIG_FAULT := TRUE;
   EnConfig := TRUE;
   AEN := TRUE;
   PV_NORM := 90.0;
   PV_SCAL := 90.0;
   AL_H3 := TRUE;
   AL_H2 := TRUE;
   AL_H1 := TRUE;
   AL_L1 := TRUE;
   AL_L2 := TRUE;
   AL_L3 := TRUE;
   SIG_OK := TRUE;
   LIM_H2 := TRUE;
   LIM_H1 := TRUE;
   MSW.VALUE := 90.0;
   MSW.EXT.AlarmWarnUnAck := TRUE;
   MSW.EXT.Operation := TRUE;
   MSW.Status := 1;
   MSW.TimeStamp := 16#3928;
   BlockInfo.Ace_Version := 80;
   BlockInfo.Ace_BuildNo := 3;
   BlockInfo.DB_Number := 5006;
   FP_PARM.Gradient_Time_ACC := 10;
   FP_PARM.OpenLoopDelay_Acc := 2;
   FP_PARM.OverRangeDelay_Acc := 2;
   ONS.SecPulse1 := TRUE;
   FIBUS_SubStatus := 16#FF;
   FIBUS_Quality := 16#FF;
   FIBUS_Limit := 16#FF;
   Result_Smooth := 90.0;
   DampXEA := 90.0;
   StatusWork := 1;
   GradientTime_Mem := 10;
   AlarmDelay_OpenLoop_Mem := 2;
   AlarmDelay_OverRange_Mem := 2;
   ScaledValue := 90.0;
   Grad_OldValue := 90.0;
   HystCalc := 1.0;
   OUT.PV_NORM := 90.0;
   OUT.PV_SCAL := 90.0;
   OUT.AL_H3 := TRUE;
   OUT.AL_H2 := TRUE;
   OUT.AL_H1 := TRUE;
   OUT.AL_L1 := TRUE;
   OUT.AL_L2 := TRUE;
   OUT.AL_L3 := TRUE;
   OUT.SIG_OK := TRUE;
   OUT.LIM_H2 := TRUE;
   OUT.LIM_H1 := TRUE;
   MSW_Status_Trans := 1;
END_DATA_BLOCK

DATA_BLOCK "_2010CV120M01I01_DB"   // DB5007
TITLE = Instance DB Analog: _2010CV120M01I01
{ S7_Optimized_Access := 'FALSE' }
AUTHOR : METIS
NAME : ANA_DB
VERSION : 8.0
// stored: InstanceOfName ACESYS_ANALOG
"ACESYS_ANALOG"
BEGIN
   FP_EN.ParentSupress := TRUE;
   FP_EN.ParentSupressUnit := TRUE;
   FP_EN.Hysteresis := TRUE;
   FP_PARM.Scale_Max := 14.0;
   FP_PARM.Grad_Pos := 0.0;
   FP_PARM.Grad_Neg := 0.0;
   FP_PARM.OpenLoopDelay_Pre := 2;
   FP_PARM.Gradient_Time_Pre := 10;
   FP_PARM.Alarm_Hyst := 1.0;
   FP_PARM.OverRangeDelay_Pre := 2;
   FP_SIM.Value_Enable := TRUE;
   FP_SIM.Gain := 1.0;
   SIG_TYPE := 1;
   IN := 3.5;
   U_RANGE := TRUE;
   O_RANGE := TRUE;
   SIG_FAULT := TRUE;
   EnConfig := TRUE;
   AEN := TRUE;
   PV_NORM := 25.0;
   PV_SCAL := 3.5;
   AL_H3 := TRUE;
   AL_H2 := TRUE;
   AL_H1 := TRUE;
   AL_L1 := TRUE;
   AL_L2 := TRUE;
   AL_L3 := TRUE;
   SIG_OK := TRUE;
   LIM_H2 := TRUE;
   LIM_H1 := TRUE;
   MSW.VALUE := 3.5;
   MSW.TRIGVALUE := 90.0;
   MSW.EXT.AlarmWarnUnAck := TRUE;
   MSW.EXT.Operation := TRUE;
   MSW.Status := 1;
   MSW.TimeStamp := 16#399B;
   BlockInfo.Ace_Version := 80;
   BlockInfo.Ace_BuildNo := 3;
   BlockInfo.DB_Number := 5007;
   FP_EN.AlarmDelay_H3 := TRUE;
   FP_PARM.Gradient_Time_ACC := 10;
   FP_PARM.AlarmLimit_H3 := 99.0;
   FP_PARM.AlarmDelay_H3_Pre := 1;
   FP_PARM.AlarmDelay_H3_Acc := 1;
   FP_PARM.OpenLoopDelay_Acc := 2;
   FP_PARM.OverRangeDelay_Acc := 2;
   ONS.SecPulse1 := TRUE;
   FIBUS_SubStatus := 16#FF;
   FIBUS_Quality := 16#FF;
   FIBUS_Limit := 16#FF;
   Result_Smooth := 25.0;
   DampXEA := 25.0;
   StatusWork := 1;
   AlarmDelay_H3_Mem := 1;
   GradientTime_Mem := 10;
   AlarmDelay_OpenLoop_Mem := 2;
   AlarmDelay_OverRange_Mem := 2;
   ScaledValue := 3.5;
   Grad_OldValue := 3.5;
   HystCalc := 0.14;
   OUT.PV_NORM := 25.0;
   OUT.PV_SCAL := 3.5;
   OUT.AL_H3 := TRUE;
   OUT.AL_H2 := TRUE;
   OUT.AL_H1 := TRUE;
   OUT.AL_L1 := TRUE;
   OUT.AL_L2 := TRUE;
   OUT.AL_L3 := TRUE;
   OUT.SIG_OK := TRUE;
   OUT.LIM_H2 := TRUE;
   OUT.LIM_H1 := TRUE;
   MSW_Status_Trans := 1;
END_DATA_BLOCK

DATA_BLOCK "_2010BF110U01I01_DB"   // DB5008
TITLE = Instance DB Analog: Current
{ S7_Optimized_Access := 'FALSE' }
AUTHOR : METIS
NAME : ANA_DB
VERSION : 8.0
// stored: InstanceOfName ACESYS_ANALOG
"ACESYS_ANALOG"
BEGIN
   FP_EN.Hysteresis := TRUE;
   FP_PARM.Scale_Max := 139.0;
   FP_PARM.Grad_Pos := 0.0;
   FP_PARM.Grad_Neg := 0.0;
   FP_PARM.OpenLoopDelay_Pre := 2;
   FP_PARM.Gradient_Time_Pre := 10;
   FP_PARM.Alarm_Hyst := 1.0;
   FP_PARM.OverRangeDelay_Pre := 2;
   FP_SIM.Value_Enable := TRUE;
   FP_SIM.Gain := 1.0;
   SIG_TYPE := 1;
   IN := 303.225;
   U_RANGE := TRUE;
   O_RANGE := TRUE;
   SIG_FAULT := TRUE;
   EnConfig := TRUE;
   AEN := TRUE;
   PV_NORM := 218.1475;
   PV_SCAL := 303.225;
   AL_H3 := TRUE;
   AL_H2 := TRUE;
   AL_H1 := TRUE;
   AL_L1 := TRUE;
   AL_L2 := TRUE;
   AL_L3 := TRUE;
   SIG_OK := TRUE;
   LIM_H2 := TRUE;
   LIM_H1 := TRUE;
   MSW.VALUE := 303.225;
   MSW.EXT.AlarmWarnUnAck := TRUE;
   MSW.EXT.Operation := TRUE;
   MSW.Status := 1;
   MSW.TimeStamp := 16#3928;
   BlockInfo.Ace_Version := 80;
   BlockInfo.Ace_BuildNo := 3;
   BlockInfo.DB_Number := 5008;
   FP_EN.U_Range_Warn := FALSE;
   FP_EN.O_Range_Warn := FALSE;
   FP_PARM.Gradient_Time_ACC := 10;
   FP_PARM.OpenLoopDelay_Acc := 2;
   FP_PARM.OverRangeDelay_Acc := 2;
   ONS.SecPulse1 := TRUE;
   FIBUS_SubStatus := 16#FF;
   FIBUS_Quality := 16#FF;
   FIBUS_Limit := 16#FF;
   Result_Smooth := 218.1475;
   DampXEA := 218.1475;
   StatusWork := 1;
   GradientTime_Mem := 10;
   AlarmDelay_OpenLoop_Mem := 2;
   AlarmDelay_OverRange_Mem := 2;
   ScaledValue := 303.225;
   Grad_OldValue := 303.225;
   HystCalc := 1.39;
   OUT.PV_NORM := 218.1475;
   OUT.PV_SCAL := 303.225;
   OUT.AL_H3 := TRUE;
   OUT.AL_H2 := TRUE;
   OUT.AL_H1 := TRUE;
   OUT.AL_L1 := TRUE;
   OUT.AL_L2 := TRUE;
   OUT.AL_L3 := TRUE;
   OUT.SIG_OK := TRUE;
   OUT.LIM_H2 := TRUE;
   OUT.LIM_H1 := TRUE;
   MSW_Status_Trans := 1;
END_DATA_BLOCK

DATA_BLOCK "_2010BF110U01J01_DB"   // DB5009
TITLE = Instance DB Analog: Power
{ S7_Optimized_Access := 'FALSE' }
AUTHOR : METIS
NAME : ANA_DB
VERSION : 8.0
// stored: InstanceOfName ACESYS_ANALOG
"ACESYS_ANALOG"
BEGIN
   FP_EN.ParentSupress := TRUE;
   FP_EN.ParentSupressUnit := TRUE;
   FP_EN.Hysteresis := TRUE;
   FP_PARM.Scale_Max := 0.01;
   FP_PARM.Grad_Pos := 0.0;
   FP_PARM.Grad_Neg := 0.0;
   FP_PARM.OpenLoopDelay_Pre := 2;
   FP_PARM.Gradient_Time_Pre := 10;
   FP_PARM.Alarm_Hyst := 1.0;
   FP_PARM.OverRangeDelay_Pre := 2;
   FP_SIM.Value_Enable := TRUE;
   FP_SIM.Gain := 1.0;
   SIG_TYPE := 1;
   IN := -15.41749;
   U_RANGE := TRUE;
   O_RANGE := TRUE;
   SIG_FAULT := TRUE;
   EnConfig := TRUE;
   AEN := TRUE;
   PV_NORM := 217.9856;
   PV_SCAL := 303.0;
   AL_H3 := TRUE;
   AL_H2 := TRUE;
   AL_H1 := TRUE;
   AL_L1 := TRUE;
   AL_L2 := TRUE;
   AL_L3 := TRUE;
   SIG_OK := TRUE;
   LIM_H2 := TRUE;
   LIM_H1 := TRUE;
   MSW.VALUE := -15.41749;
   MSW.EXT.AlarmWarnUnAck := TRUE;
   MSW.EXT.Operation := TRUE;
   MSW.Status := 1;
   MSW.TimeStamp := 16#3928;
   BlockInfo.Ace_Version := 80;
   BlockInfo.Ace_BuildNo := 3;
   BlockInfo.DB_Number := 5006;
   FP_PARM.Gradient_Time_ACC := 10;
   FP_PARM.OpenLoopDelay_Acc := 2;
   FP_PARM.OverRangeDelay_Acc := 2;
   ONS.SecPulse2 := TRUE;
   FIBUS_SubStatus := 16#FF;
   FIBUS_Quality := 16#FF;
   FIBUS_Limit := 16#FF;
   Result_Smooth := -154174.9;
   DampXEA := -154174.9;
   StatusWork := 1;
   GradientTime_Mem := 10;
   AlarmDelay_OpenLoop_Mem := 2;
   AlarmDelay_OverRange_Mem := 2;
   ScaledValue := -15.41749;
   Grad_OldValue := -15.41749;
   HystCalc := 0.0001;
   OUT.PV_NORM := -154174.9;
   OUT.PV_SCAL := -15.41749;
   OUT.AL_H3 := TRUE;
   OUT.AL_H2 := TRUE;
   OUT.AL_H1 := TRUE;
   OUT.AL_L1 := TRUE;
   OUT.AL_L2 := TRUE;
   OUT.AL_L3 := TRUE;
   OUT.SIG_OK := TRUE;
   OUT.LIM_L1 := TRUE;
   OUT.LIM_L2 := TRUE;
   MSW_Status_Trans := 1;
END_DATA_BLOCK

DATA_BLOCK "_2010BF110U01S01_DB"   // DB5010
TITLE = Instance DB Analog: Speed
{ S7_Optimized_Access := 'FALSE' }
AUTHOR : METIS
NAME : ANA_DB
VERSION : 8.0
// stored: InstanceOfName ACESYS_ANALOG
"ACESYS_ANALOG"
BEGIN
   FP_EN.ParentSupress := TRUE;
   FP_EN.ParentSupressUnit := TRUE;
   FP_EN.Hysteresis := TRUE;
   FP_PARM.Grad_Pos := 0.0;
   FP_PARM.Grad_Neg := 0.0;
   FP_PARM.OpenLoopDelay_Pre := 2;
   FP_PARM.Gradient_Time_Pre := 10;
   FP_PARM.Alarm_Hyst := 1.0;
   FP_PARM.OverRangeDelay_Pre := 2;
   FP_SIM.Value_Enable := TRUE;
   FP_SIM.Gain := 1.0;
   IN := 30.0;
   U_RANGE := TRUE;
   O_RANGE := TRUE;
   SIG_FAULT := TRUE;
   EnConfig := TRUE;
   AEN := TRUE;
   PV_NORM := 30.0;
   PV_SCAL := 30.0;
   AL_H3 := TRUE;
   AL_H2 := TRUE;
   AL_H1 := TRUE;
   AL_L1 := TRUE;
   AL_L2 := TRUE;
   AL_L3 := TRUE;
   SIG_OK := TRUE;
   LIM_H2 := TRUE;
   LIM_H1 := TRUE;
   MSW.VALUE := 30.0;
   MSW.EXT.AlarmWarnUnAck := TRUE;
   MSW.EXT.Operation := TRUE;
   MSW.Status := 1;
   MSW.TimeStamp := 16#3928;
   BlockInfo.Ace_Version := 80;
   BlockInfo.Ace_BuildNo := 3;
   BlockInfo.DB_Number := 5010;
   FP_PARM.Gradient_Time_ACC := 10;
   FP_PARM.OpenLoopDelay_Acc := 2;
   FP_PARM.OverRangeDelay_Acc := 2;
   ONS.SecPulse1 := TRUE;
   FIBUS_SubStatus := 16#FF;
   FIBUS_Quality := 16#FF;
   FIBUS_Limit := 16#FF;
   Result_Smooth := 30.0;
   DampXEA := 30.0;
   StatusWork := 1;
   GradientTime_Mem := 10;
   AlarmDelay_OpenLoop_Mem := 2;
   AlarmDelay_OverRange_Mem := 2;
   ScaledValue := 30.0;
   Grad_OldValue := 30.0;
   HystCalc := 1.0;
   OUT.PV_NORM := 30.0;
   OUT.PV_SCAL := 30.0;
   OUT.AL_H3 := TRUE;
   OUT.AL_H2 := TRUE;
   OUT.AL_H1 := TRUE;
   OUT.AL_L1 := TRUE;
   OUT.AL_L2 := TRUE;
   OUT.AL_L3 := TRUE;
   OUT.SIG_OK := TRUE;
   OUT.LIM_H2 := TRUE;
   OUT.LIM_H1 := TRUE;
   MSW_Status_Trans := 1;
END_DATA_BLOCK

DATA_BLOCK "_2010BF110U01GT01_DB"   // DB5011
TITLE = Instance DB Analog:
{ S7_Optimized_Access := 'FALSE' }
AUTHOR : METIS
NAME : ANA_DB
VERSION : 8.0
// stored: InstanceOfName ACESYS_ANALOG
"ACESYS_ANALOG"
BEGIN
   FP_EN.ParentSupress := TRUE;
   FP_EN.ParentSupressUnit := TRUE;
   FP_EN.Hysteresis := TRUE;
   FP_PARM.Scale_Max := 0.01;
   FP_PARM.Grad_Pos := 0.0;
   FP_PARM.Grad_Neg := 0.0;
   FP_PARM.OpenLoopDelay_Pre := 2;
   FP_PARM.Gradient_Time_Pre := 10;
   FP_PARM.Alarm_Hyst := 1.0;
   FP_PARM.OverRangeDelay_Pre := 2;
   FP_SIM.Value_Enable := TRUE;
   FP_SIM.Gain := 1.0;
   SIG_TYPE := 1;
   IN := 0.04701968;
   U_RANGE := TRUE;
   O_RANGE := TRUE;
   SIG_FAULT := TRUE;
   EnConfig := TRUE;
   AEN := TRUE;
   PV_NORM := -154174.9;
   PV_SCAL := -15.41749;
   AL_H3 := TRUE;
   AL_H2 := TRUE;
   AL_H1 := TRUE;
   AL_L1 := TRUE;
   AL_L2 := TRUE;
   AL_L3 := TRUE;
   SIG_OK := TRUE;
   LIM_L1 := TRUE;
   LIM_L2 := TRUE;
   MSW.VALUE := -15.41749;
   MSW.EXT.AlarmWarnUnAck := TRUE;
   MSW.EXT.Operation := TRUE;
   MSW.Status := 1;
   MSW.TimeStamp := 16#3928;
   BlockInfo.Ace_Version := 80;
   BlockInfo.Ace_BuildNo := 3;
   BlockInfo.DB_Number := 5006;
   FP_PARM.Gradient_Time_ACC := 10;
   FP_PARM.OpenLoopDelay_Acc := 2;
   FP_PARM.OverRangeDelay_Acc := 2;
   ONS.SecPulse2 := TRUE;
   FIBUS_SubStatus := 16#FF;
   FIBUS_Quality := 16#FF;
   FIBUS_Limit := 16#FF;
   Result_Smooth := -154174.9;
   DampXEA := -154174.9;
   StatusWork := 1;
   GradientTime_Mem := 10;
   AlarmDelay_OpenLoop_Mem := 2;
   AlarmDelay_OverRange_Mem := 2;
   ScaledValue := -15.41749;
   Grad_OldValue := -15.41749;
   HystCalc := 0.0001;
   OUT.PV_NORM := -154174.9;
   OUT.PV_SCAL := -15.41749;
   OUT.AL_H3 := TRUE;
   OUT.AL_H2 := TRUE;
   OUT.AL_H1 := TRUE;
   OUT.AL_L1 := TRUE;
   OUT.AL_L2 := TRUE;
   OUT.AL_L3 := TRUE;
   OUT.SIG_OK := TRUE;
   OUT.LIM_L1 := TRUE;
   OUT.LIM_L2 := TRUE;
   MSW_Status_Trans := 1;
END_DATA_BLOCK

DATA_BLOCK "_2010BF110U01S02_DB"   // DB5012
TITLE = Instance DB Analog: Speed
{ S7_Optimized_Access := 'FALSE' }
AUTHOR : METIS
NAME : ANA_DB
VERSION : 8.0
// stored: InstanceOfName ACESYS_ANALOG
"ACESYS_ANALOG"
BEGIN
   FP_EN.ParentSupress := TRUE;
   FP_EN.ParentSupressUnit := TRUE;
   FP_EN.Hysteresis := TRUE;
   FP_PARM.Scale_Max := 0.01;
   FP_PARM.Grad_Pos := 0.0;
   FP_PARM.Grad_Neg := 0.0;
   FP_PARM.OpenLoopDelay_Pre := 2;
   FP_PARM.Gradient_Time_Pre := 10;
   FP_PARM.Alarm_Hyst := 1.0;
   FP_PARM.OverRangeDelay_Pre := 2;
   FP_SIM.Value_Enable := TRUE;
   FP_SIM.Gain := 1.0;
   SIG_TYPE := 1;
   IN := 283.5;
   U_RANGE := TRUE;
   O_RANGE := TRUE;
   SIG_FAULT := TRUE;
   EnConfig := TRUE;
   AEN := TRUE;
   PV_NORM := 2835000.0;
   PV_SCAL := 283.5;
   AL_H3 := TRUE;
   AL_H2 := TRUE;
   AL_H1 := TRUE;
   AL_L1 := TRUE;
   AL_L2 := TRUE;
   AL_L3 := TRUE;
   SIG_OK := TRUE;
   LIM_H2 := TRUE;
   LIM_H1 := TRUE;
   MSW.VALUE := 283.5;
   MSW.EXT.AlarmWarnUnAck := TRUE;
   MSW.EXT.Operation := TRUE;
   MSW.Status := 1;
   MSW.TimeStamp := 16#3928;
   BlockInfo.Ace_Version := 80;
   BlockInfo.Ace_BuildNo := 3;
   BlockInfo.DB_Number := 5012;
   FP_PARM.Gradient_Time_ACC := 10;
   FP_PARM.OpenLoopDelay_Acc := 2;
   FP_PARM.OverRangeDelay_Acc := 2;
   ONS.SecPulse2 := TRUE;
   FIBUS_SubStatus := 16#FF;
   FIBUS_Quality := 16#FF;
   FIBUS_Limit := 16#FF;
   Result_Smooth := 2835000.0;
   DampXEA := 2835000.0;
   Sec_Pulse := TRUE;
   StatusWork := 1;
   GradientTime_Mem := 10;
   AlarmDelay_OpenLoop_Mem := 2;
   AlarmDelay_OverRange_Mem := 2;
   ScaledValue := 283.5;
   Grad_OldValue := 283.5;
   HystCalc := 0.0001;
   OUT.PV_NORM := 2835000.0;
   OUT.PV_SCAL := 283.5;
   OUT.AL_H3 := TRUE;
   OUT.AL_H2 := TRUE;
   OUT.AL_H1 := TRUE;
   OUT.AL_L1 := TRUE;
   OUT.AL_L2 := TRUE;
   OUT.AL_L3 := TRUE;
   OUT.SIG_OK := TRUE;
   OUT.LIM_H2 := TRUE;
   OUT.LIM_H1 := TRUE;
   MSW_Status_Trans := 1;
END_DATA_BLOCK

DATA_BLOCK "_2010SC130U01I01_DB"   // DB5013
TITLE = Instance DB Analog: Current
{ S7_Optimized_Access := 'FALSE' }
AUTHOR : METIS
NAME : ANA_DB
VERSION : 8.0
// stored: InstanceOfName ACESYS_ANALOG
"ACESYS_ANALOG"
BEGIN
   FP_EN.Hysteresis := TRUE;
   FP_PARM.Scale_Max := 134.0;
   FP_PARM.Grad_Pos := 0.0;
   FP_PARM.Grad_Neg := 0.0;
   FP_PARM.OpenLoopDelay_Pre := 2;
   FP_PARM.Gradient_Time_Pre := 10;
   FP_PARM.Alarm_Hyst := 1.0;
   FP_PARM.OverRangeDelay_Pre := 2;
   FP_SIM.Value_Enable := TRUE;
   FP_SIM.Gain := 1.0;
   SIG_TYPE := 1;
   IN := 304.35;
   U_RANGE := TRUE;
   O_RANGE := TRUE;
   SIG_FAULT := TRUE;
   EnConfig := TRUE;
   AEN := TRUE;
   PV_NORM := 227.1269;
   PV_SCAL := 304.35;
   AL_H3 := TRUE;
   AL_H2 := TRUE;
   AL_H1 := TRUE;
   AL_L1 := TRUE;
   AL_L2 := TRUE;
   AL_L3 := TRUE;
   SIG_OK := TRUE;
   LIM_H2 := TRUE;
   LIM_H1 := TRUE;
   MSW.VALUE := 304.35;
   MSW.EXT.AlarmWarnUnAck := TRUE;
   MSW.EXT.Operation := TRUE;
   MSW.Status := 1;
   MSW.TimeStamp := 16#3928;
   BlockInfo.Ace_Version := 80;
   BlockInfo.Ace_BuildNo := 3;
   BlockInfo.DB_Number := 5013;
   FP_PARM.Gradient_Time_ACC := 10;
   FP_PARM.OpenLoopDelay_Acc := 2;
   FP_PARM.OverRangeDelay_Acc := 2;
   ONS.SecPulse2 := TRUE;
   FIBUS_SubStatus := 16#FF;
   FIBUS_Quality := 16#FF;
   FIBUS_Limit := 16#FF;
   Result_Smooth := 227.1269;
   DampXEA := 227.1269;
   StatusWork := 1;
   GradientTime_Mem := 10;
   AlarmDelay_OpenLoop_Mem := 2;
   AlarmDelay_OverRange_Mem := 2;
   ScaledValue := 304.35;
   Grad_OldValue := 304.35;
   HystCalc := 1.34;
   OUT.PV_NORM := 227.1269;
   OUT.PV_SCAL := 304.35;
   OUT.AL_H3 := TRUE;
   OUT.AL_H2 := TRUE;
   OUT.AL_H1 := TRUE;
   OUT.AL_L1 := TRUE;
   OUT.AL_L2 := TRUE;
   OUT.AL_L3 := TRUE;
   OUT.SIG_OK := TRUE;
   OUT.LIM_H2 := TRUE;
   OUT.LIM_H1 := TRUE;
   MSW_Status_Trans := 1;
END_DATA_BLOCK

DATA_BLOCK "_2010SC130U01J01_DB"   // DB5014
TITLE = Instance DB Analog: Power
{ S7_Optimized_Access := 'FALSE' }
AUTHOR : METIS
NAME : ANA_DB
VERSION : 8.0
// stored: InstanceOfName ACESYS_ANALOG
"ACESYS_ANALOG"
BEGIN
   FP_EN.ParentSupress := TRUE;
   FP_EN.ParentSupressUnit := TRUE;
   FP_EN.Hysteresis := TRUE;
   FP_PARM.Scale_Max := 0.01;
   FP_PARM.Grad_Pos := 0.0;
   FP_PARM.Grad_Neg := 0.0;
   FP_PARM.OpenLoopDelay_Pre := 2;
   FP_PARM.Gradient_Time_Pre := 10;
   FP_PARM.Alarm_Hyst := 1.0;
   FP_PARM.OverRangeDelay_Pre := 2;
   FP_SIM.Value_Enable := TRUE;
   FP_SIM.Gain := 1.0;
   SIG_TYPE := 1;
   IN := -15.41749;
   U_RANGE := TRUE;
   O_RANGE := TRUE;
   SIG_FAULT := TRUE;
   EnConfig := TRUE;
   AEN := TRUE;
   PV_NORM := 227.1269;
   PV_SCAL := 304.35;
   AL_H3 := TRUE;
   AL_H2 := TRUE;
   AL_H1 := TRUE;
   AL_L1 := TRUE;
   AL_L2 := TRUE;
   AL_L3 := TRUE;
   SIG_OK := TRUE;
   LIM_H2 := TRUE;
   LIM_H1 := TRUE;
   MSW.VALUE := -15.41749;
   MSW.EXT.AlarmWarnUnAck := TRUE;
   MSW.EXT.Operation := TRUE;
   MSW.Status := 1;
   MSW.TimeStamp := 16#3928;
   BlockInfo.Ace_Version := 80;
   BlockInfo.Ace_BuildNo := 3;
   BlockInfo.DB_Number := 5006;
   FP_PARM.Gradient_Time_ACC := 10;
   FP_PARM.OpenLoopDelay_Acc := 2;
   FP_PARM.OverRangeDelay_Acc := 2;
   ONS.SecPulse2 := TRUE;
   FIBUS_SubStatus := 16#FF;
   FIBUS_Quality := 16#FF;
   FIBUS_Limit := 16#FF;
   Result_Smooth := -154174.9;
   DampXEA := -154174.9;
   StatusWork := 1;
   GradientTime_Mem := 10;
   AlarmDelay_OpenLoop_Mem := 2;
   AlarmDelay_OverRange_Mem := 2;
   ScaledValue := -15.41749;
   Grad_OldValue := -15.41749;
   HystCalc := 0.0001;
   OUT.PV_NORM := -154174.9;
   OUT.PV_SCAL := -15.41749;
   OUT.AL_H3 := TRUE;
   OUT.AL_H2 := TRUE;
   OUT.AL_H1 := TRUE;
   OUT.AL_L1 := TRUE;
   OUT.AL_L2 := TRUE;
   OUT.AL_L3 := TRUE;
   OUT.SIG_OK := TRUE;
   OUT.LIM_L1 := TRUE;
   OUT.LIM_L2 := TRUE;
   MSW_Status_Trans := 1;
END_DATA_BLOCK

DATA_BLOCK "_2010SC130U01S01_DB"   // DB5015
TITLE = Instance DB Analog: Speed
{ S7_Optimized_Access := 'FALSE' }
AUTHOR : METIS
NAME : ANA_DB
VERSION : 8.0
// stored: InstanceOfName ACESYS_ANALOG
"ACESYS_ANALOG"
BEGIN
   FP_EN.Hysteresis := TRUE;
   FP_PARM.Grad_Pos := 0.0;
   FP_PARM.Grad_Neg := 0.0;
   FP_PARM.OpenLoopDelay_Pre := 2;
   FP_PARM.Gradient_Time_Pre := 10;
   FP_PARM.Alarm_Hyst := 1.0;
   FP_PARM.OverRangeDelay_Pre := 2;
   FP_SIM.Value_Enable := TRUE;
   FP_SIM.Gain := 1.0;
   IN := 100.0;
   U_RANGE := TRUE;
   O_RANGE := TRUE;
   SIG_FAULT := TRUE;
   EnConfig := TRUE;
   AEN := TRUE;
   PV_NORM := 100.0;
   PV_SCAL := 100.0;
   AL_H3 := TRUE;
   AL_H2 := TRUE;
   AL_H1 := TRUE;
   AL_L1 := TRUE;
   AL_L2 := TRUE;
   AL_L3 := TRUE;
   SIG_OK := TRUE;
   LIM_H2 := TRUE;
   LIM_H1 := TRUE;
   MSW.VALUE := 100.0;
   MSW.EXT.AlarmWarnUnAck := TRUE;
   MSW.EXT.Operation := TRUE;
   MSW.Status := 1;
   MSW.TimeStamp := 16#3928;
   BlockInfo.Ace_Version := 80;
   BlockInfo.Ace_BuildNo := 3;
   BlockInfo.DB_Number := 5015;
   FP_PARM.Gradient_Time_ACC := 10;
   FP_PARM.OpenLoopDelay_Acc := 2;
   FP_PARM.OverRangeDelay_Acc := 2;
   ONS.SecPulse2 := TRUE;
   FIBUS_SubStatus := 16#FF;
   FIBUS_Quality := 16#FF;
   FIBUS_Limit := 16#FF;
   Result_Smooth := 100.0;
   DampXEA := 100.0;
   StatusWork := 1;
   GradientTime_Mem := 10;
   AlarmDelay_OpenLoop_Mem := 2;
   AlarmDelay_OverRange_Mem := 2;
   ScaledValue := 100.0;
   Grad_OldValue := 100.0;
   HystCalc := 1.0;
   OUT.PV_NORM := 100.0;
   OUT.PV_SCAL := 100.0;
   OUT.AL_H3 := TRUE;
   OUT.AL_H2 := TRUE;
   OUT.AL_H1 := TRUE;
   OUT.AL_L1 := TRUE;
   OUT.AL_L2 := TRUE;
   OUT.AL_L3 := TRUE;
   OUT.SIG_OK := TRUE;
   OUT.LIM_H2 := TRUE;
   OUT.LIM_H1 := TRUE;
   MSW_Status_Trans := 1;
END_DATA_BLOCK

DATA_BLOCK "_2010CR150M01I01_DB"   // DB5016
TITLE = Instance DB Analog: Current
{ S7_Optimized_Access := 'FALSE' }
AUTHOR : METIS
NAME : ANA_DB
VERSION : 8.0
// stored: InstanceOfName ACESYS_ANALOG
"ACESYS_ANALOG"
BEGIN
   FP_EN.Hysteresis := TRUE;
   FP_PARM.Scale_Max := 2065.0;
   FP_PARM.Grad_Pos := 0.0;
   FP_PARM.Grad_Neg := 0.0;
   FP_PARM.OpenLoopDelay_Pre := 2;
   FP_PARM.Gradient_Time_Pre := 10;
   FP_PARM.Alarm_Hyst := 1.0;
   FP_PARM.OverRangeDelay_Pre := 2;
   FP_SIM.Value_Enable := TRUE;
   FP_SIM.Gain := 1.0;
   IN := 9.917535;
   U_RANGE := TRUE;
   O_RANGE := TRUE;
   SIG_FAULT := TRUE;
   EnConfig := TRUE;
   AEN := TRUE;
   PV_NORM := 6.993275;
   PV_SCAL := 144.4111;
   AL_H3 := TRUE;
   AL_H2 := TRUE;
   AL_H1 := TRUE;
   AL_L1 := TRUE;
   AL_L2 := TRUE;
   AL_L3 := TRUE;
   SIG_OK := TRUE;
   LIM_H1 := TRUE;
   MSW.VALUE := 144.4111;
   MSW.TRIGVALUE := 250.3007;
   MSW.EXT.AlarmWarnUnAck := TRUE;
   MSW.EXT.Operation := TRUE;
   MSW.Status := 1;
   MSW.TimeStamp := 16#0536;
   BlockInfo.Ace_Version := 80;
   BlockInfo.Ace_BuildNo := 3;
   BlockInfo.DB_Number := 5016;
   FP_EN.Damping := TRUE;
   FP_EN.Alarm_H2 := TRUE;
   FP_EN.Alarm_H1 := TRUE;
   FP_EN.AlarmDelay_H2 := TRUE;
   FP_EN.AlarmDelay_H1 := TRUE;
   FP_PARM.DampingTime := 4;
   FP_PARM.Gradient_Time_ACC := 10;
   FP_PARM.AlarmLimit_H3 := 1000.0;
   FP_PARM.AlarmLimit_H2 := 400.0;
   FP_PARM.AlarmLimit_H1 := 320.0;
   FP_PARM.AlarmDelay_H2_Pre := 10;
   FP_PARM.AlarmDelay_H2_Acc := 10;
   FP_PARM.AlarmDelay_H1_Pre := 5;
   FP_PARM.AlarmDelay_H1_Acc := 5;
   FP_PARM.OpenLoopDelay_Acc := 2;
   FP_PARM.OverRangeDelay_Acc := 2;
   FP_PARM.AuxLimit_H2_Value := 400.0;
   ONS.SecPulse2 := TRUE;
   ONS.DampingOn := TRUE;
   FIBUS_SubStatus := 16#FF;
   FIBUS_Quality := 16#FF;
   FIBUS_Limit := 16#FF;
   Result_Smooth := 6.993275;
   DampXA := 6.993275;
   DampXEA := 7.227242;
   StatusWork := 1;
   AlarmDelay_H2_Mem := 10;
   AlarmDelay_H1_Mem := 5;
   GradientTime_Mem := 10;
   AlarmDelay_OpenLoop_Mem := 2;
   AlarmDelay_OverRange_Mem := 2;
   ScaledValue := 144.4111;
   Grad_OldValue := 144.4111;
   HystCalc := 20.65;
   OUT.PV_NORM := 6.993275;
   OUT.PV_SCAL := 144.4111;
   OUT.AL_H3 := TRUE;
   OUT.AL_H2 := TRUE;
   OUT.AL_H1 := TRUE;
   OUT.AL_L1 := TRUE;
   OUT.AL_L2 := TRUE;
   OUT.AL_L3 := TRUE;
   OUT.SIG_OK := TRUE;
   OUT.LIM_H1 := TRUE;
   MSW_Status_Trans := 1;
END_DATA_BLOCK

DATA_BLOCK "_2010CR150M01L01_DB"   // DB5017
TITLE = Instance DB Analog: Speed
{ S7_Optimized_Access := 'FALSE' }
AUTHOR : METIS
NAME : ANA_DB
VERSION : 8.0
// stored: InstanceOfName ACESYS_ANALOG
"ACESYS_ANALOG"
BEGIN
   FP_EN.Hysteresis := TRUE;
   FP_PARM.Grad_Pos := 0.0;
   FP_PARM.Grad_Neg := 0.0;
   FP_PARM.OpenLoopDelay_Pre := 2;
   FP_PARM.Gradient_Time_Pre := 10;
   FP_PARM.Alarm_Hyst := 1.0;
   FP_PARM.OverRangeDelay_Pre := 2;
   FP_SIM.Value_Enable := TRUE;
   FP_SIM.Gain := 1.0;
   IN := -118.5185;
   U_RANGE := TRUE;
   O_RANGE := TRUE;
   SIG_FAULT := TRUE;
   EnConfig := TRUE;
   AEN := TRUE;
   PV_NORM := -118.5185;
   PV_SCAL := -118.5185;
   AL_H3 := TRUE;
   AL_H2 := TRUE;
   AL_H1 := TRUE;
   AL_L1 := TRUE;
   AL_L2 := TRUE;
   AL_L3 := TRUE;
   SIG_OK := TRUE;
   LIM_L1 := TRUE;
   LIM_L2 := TRUE;
   MSW.VALUE := -118.5185;
   MSW.TRIGVALUE := -118.5185;
   MSW.EXT.AlarmWarnUnAck := TRUE;
   MSW.EXT.Operation := TRUE;
   MSW.Status := 1;
   MSW.TimeStamp := 16#7334;
   BlockInfo.Ace_Version := 80;
   BlockInfo.Ace_BuildNo := 3;
   BlockInfo.DB_Number := 5017;
   FP_EN.Alarm_H2 := TRUE;
   FP_PARM.Force_Value := 90.0;
   FP_PARM.Gradient_Time_ACC := 10;
   FP_PARM.AlarmLimit_H2 := 80.0;
   FP_PARM.OpenLoopDelay_Acc := 2;
   FP_PARM.OverRangeDelay_Acc := 2;
   ONS.SecPulse2 := TRUE;
   FIBUS_SubStatus := 16#FF;
   FIBUS_Quality := 16#FF;
   FIBUS_Limit := 16#FF;
   Result_Smooth := -118.5185;
   DampXEA := -118.5185;
   StatusWork := 1;
   GradientTime_Mem := 10;
   AlarmDelay_OpenLoop_Mem := 2;
   AlarmDelay_OverRange_Mem := 2;
   ScaledValue := -118.5185;
   Grad_OldValue := -118.5185;
   HystCalc := 1.0;
   OUT.PV_NORM := -118.5185;
   OUT.PV_SCAL := -118.5185;
   OUT.AL_H3 := TRUE;
   OUT.AL_H2 := TRUE;
   OUT.AL_H1 := TRUE;
   OUT.AL_L1 := TRUE;
   OUT.AL_L2 := TRUE;
   OUT.AL_L3 := TRUE;
   OUT.SIG_OK := TRUE;
   OUT.LIM_L1 := TRUE;
   OUT.LIM_L2 := TRUE;
   MSW_Status_Trans := 1;
END_DATA_BLOCK

DATA_BLOCK "_2010CR150A01T01_DB"   // DB5018
TITLE = Instance DB Analog: Temp
{ S7_Optimized_Access := 'FALSE' }
AUTHOR : METIS
NAME : ANA_DB
VERSION : 8.0
// stored: InstanceOfName ACESYS_ANALOG
"ACESYS_ANALOG"
BEGIN
   FP_EN.ParentSupress := TRUE;
   FP_EN.ParentSupressUnit := TRUE;
   FP_EN.Hysteresis := TRUE;
   FP_PARM.Scale_Max := 200.0;
   FP_PARM.Grad_Pos := 0.0;
   FP_PARM.Grad_Neg := 0.0;
   FP_PARM.OpenLoopDelay_Pre := 2;
   FP_PARM.Gradient_Time_Pre := 10;
   FP_PARM.Alarm_Hyst := 1.0;
   FP_PARM.OverRangeDelay_Pre := 2;
   FP_SIM.Value_Enable := TRUE;
   FP_SIM.Gain := 1.0;
   IN := 40.84925;
   U_RANGE := TRUE;
   O_RANGE := TRUE;
   SIG_FAULT := TRUE;
   EnConfig := TRUE;
   AEN := TRUE;
   PV_NORM := 40.84925;
   PV_SCAL := 52.12312;
   AL_H3 := TRUE;
   AL_H2 := TRUE;
   AL_H1 := TRUE;
   AL_L1 := TRUE;
   AL_L2 := TRUE;
   AL_L3 := TRUE;
   SIG_OK := TRUE;
   LIM_H2 := TRUE;
   LIM_H1 := TRUE;
   MSW.VALUE := 52.12312;
   MSW.TRIGVALUE := -84.81264;
   MSW.EXT.AlarmWarnUnAck := TRUE;
   MSW.EXT.Operation := TRUE;
   MSW.Status := 1;
   MSW.TimeStamp := 16#72EF;
   BlockInfo.Ace_Version := 80;
   BlockInfo.Ace_BuildNo := 3;
   BlockInfo.DB_Number := 5018;
   FP_EN.Alarm_H2 := TRUE;
   FP_EN.Alarm_H1 := TRUE;
   FP_PARM.Scale_Min := -50.0;
   FP_PARM.Gradient_Time_ACC := 10;
   FP_PARM.AlarmLimit_H2 := 85.0;
   FP_PARM.AlarmLimit_H1 := 80.0;
   FP_PARM.AlarmDelay_H2_Pre := 5;
   FP_PARM.AlarmDelay_H2_Acc := 5;
   FP_PARM.AlarmDelay_H1_Pre := 5;
   FP_PARM.AlarmDelay_H1_Acc := 5;
   FP_PARM.OpenLoopDelay_Acc := 2;
   FP_PARM.OverRangeDelay_Acc := 2;
   ONS.SecPulse2 := TRUE;
   FIBUS_SubStatus := 16#FF;
   FIBUS_Quality := 16#FF;
   FIBUS_Limit := 16#FF;
   Result_Smooth := 40.84925;
   DampXEA := 40.84925;
   StatusWork := 1;
   AlarmDelay_H2_Mem := 5;
   AlarmDelay_H1_Mem := 5;
   GradientTime_Mem := 10;
   AlarmDelay_OpenLoop_Mem := 2;
   AlarmDelay_OverRange_Mem := 2;
   ScaledValue := 52.12312;
   Grad_OldValue := 52.12312;
   HystCalc := 2.5;
   OUT.PV_NORM := 40.84925;
   OUT.PV_SCAL := 52.12312;
   OUT.AL_H3 := TRUE;
   OUT.AL_H2 := TRUE;
   OUT.AL_H1 := TRUE;
   OUT.AL_L1 := TRUE;
   OUT.AL_L2 := TRUE;
   OUT.AL_L3 := TRUE;
   OUT.SIG_OK := TRUE;
   OUT.LIM_H2 := TRUE;
   OUT.LIM_H1 := TRUE;
   MSW_Status_Trans := 1;
END_DATA_BLOCK

DATA_BLOCK "_2010CR150A01T02_DB"   // DB5019
TITLE = Instance DB Analog: Temp
{ S7_Optimized_Access := 'FALSE' }
AUTHOR : METIS
NAME : ANA_DB
VERSION : 8.0
// stored: InstanceOfName ACESYS_ANALOG
"ACESYS_ANALOG"
BEGIN
   FP_EN.ParentSupress := TRUE;
   FP_EN.ParentSupressUnit := TRUE;
   FP_EN.Hysteresis := TRUE;
   FP_PARM.Scale_Max := 200.0;
   FP_PARM.Grad_Pos := 0.0;
   FP_PARM.Grad_Neg := 0.0;
   FP_PARM.OpenLoopDelay_Pre := 2;
   FP_PARM.Gradient_Time_Pre := 10;
   FP_PARM.Alarm_Hyst := 1.0;
   FP_PARM.OverRangeDelay_Pre := 2;
   FP_SIM.Value_Enable := TRUE;
   FP_SIM.Gain := 1.0;
   IN := 40.80946;
   U_RANGE := TRUE;
   O_RANGE := TRUE;
   SIG_FAULT := TRUE;
   EnConfig := TRUE;
   AEN := TRUE;
   PV_NORM := 40.80946;
   PV_SCAL := 52.02366;
   AL_H3 := TRUE;
   AL_H2 := TRUE;
   AL_H1 := TRUE;
   AL_L1 := TRUE;
   AL_L2 := TRUE;
   AL_L3 := TRUE;
   SIG_OK := TRUE;
   LIM_H2 := TRUE;
   LIM_H1 := TRUE;
   MSW.VALUE := 52.02366;
   MSW.TRIGVALUE := -71.1046;
   MSW.EXT.AlarmWarnUnAck := TRUE;
   MSW.EXT.Operation := TRUE;
   MSW.Status := 1;
   MSW.TimeStamp := 16#72F7;
   BlockInfo.Ace_Version := 80;
   BlockInfo.Ace_BuildNo := 3;
   BlockInfo.DB_Number := 5019;
   FP_EN.Alarm_H2 := TRUE;
   FP_EN.Alarm_H1 := TRUE;
   FP_EN.AlarmDelay_H2 := TRUE;
   FP_EN.AlarmDelay_H1 := TRUE;
   FP_PARM.Scale_Min := -50.0;
   FP_PARM.Gradient_Time_ACC := 10;
   FP_PARM.AlarmLimit_H2 := 85.0;
   FP_PARM.AlarmLimit_H1 := 80.0;
   FP_PARM.AlarmDelay_H2_Pre := 5;
   FP_PARM.AlarmDelay_H2_Acc := 5;
   FP_PARM.AlarmDelay_H1_Pre := 5;
   FP_PARM.AlarmDelay_H1_Acc := 5;
   FP_PARM.OpenLoopDelay_Acc := 2;
   FP_PARM.OverRangeDelay_Acc := 2;
   ONS.SecPulse2 := TRUE;
   FIBUS_SubStatus := 16#FF;
   FIBUS_Quality := 16#FF;
   FIBUS_Limit := 16#FF;
   Result_Smooth := 40.80946;
   DampXEA := 40.80946;
   StatusWork := 1;
   AlarmDelay_H2_Mem := 5;
   AlarmDelay_H1_Mem := 5;
   GradientTime_Mem := 10;
   AlarmDelay_OpenLoop_Mem := 2;
   AlarmDelay_OverRange_Mem := 2;
   ScaledValue := 52.02366;
   Grad_OldValue := 52.02366;
   HystCalc := 2.5;
   OUT.PV_NORM := 40.80946;
   OUT.PV_SCAL := 52.02366;
   OUT.AL_H3 := TRUE;
   OUT.AL_H2 := TRUE;
   OUT.AL_H1 := TRUE;
   OUT.AL_L1 := TRUE;
   OUT.AL_L2 := TRUE;
   OUT.AL_L3 := TRUE;
   OUT.SIG_OK := TRUE;
   OUT.LIM_H2 := TRUE;
   OUT.LIM_H1 := TRUE;
   MSW_Status_Trans := 1;
END_DATA_BLOCK

DATA_BLOCK "_2010CR150A01T03_DB"   // DB5020
TITLE = Instance DB Analog: Temp
{ S7_Optimized_Access := 'FALSE' }
AUTHOR : METIS
NAME : ANA_DB
VERSION : 8.0
// stored: InstanceOfName ACESYS_ANALOG
"ACESYS_ANALOG"
BEGIN
   FP_EN.ParentSupress := TRUE;
   FP_EN.ParentSupressUnit := TRUE;
   FP_EN.Hysteresis := TRUE;
   FP_PARM.Scale_Max := 200.0;
   FP_PARM.Grad_Pos := 0.0;
   FP_PARM.Grad_Neg := 0.0;
   FP_PARM.OpenLoopDelay_Pre := 2;
   FP_PARM.Gradient_Time_Pre := 10;
   FP_PARM.Alarm_Hyst := 1.0;
   FP_PARM.OverRangeDelay_Pre := 2;
   FP_SIM.Value_Enable := TRUE;
   FP_SIM.Gain := 1.0;
   IN := 45.74653;
   U_RANGE := TRUE;
   O_RANGE := TRUE;
   SIG_FAULT := TRUE;
   EnConfig := TRUE;
   AEN := TRUE;
   PV_NORM := 45.74653;
   PV_SCAL := 64.36632;
   AL_H3 := TRUE;
   AL_H2 := TRUE;
   AL_H1 := TRUE;
   AL_L1 := TRUE;
   AL_L2 := TRUE;
   AL_L3 := TRUE;
   SIG_OK := TRUE;
   LIM_H2 := TRUE;
   LIM_H1 := TRUE;
   MSW.VALUE := 64.36632;
   MSW.TRIGVALUE := -69.39561;
   MSW.EXT.AlarmWarnUnAck := TRUE;
   MSW.EXT.Operation := TRUE;
   MSW.Status := 1;
   MSW.TimeStamp := 16#72FC;
   BlockInfo.Ace_Version := 80;
   BlockInfo.Ace_BuildNo := 3;
   BlockInfo.DB_Number := 5020;
   FP_EN.Alarm_H2 := TRUE;
   FP_EN.Alarm_H1 := TRUE;
   FP_EN.AlarmDelay_H2 := TRUE;
   FP_EN.AlarmDelay_H1 := TRUE;
   FP_PARM.Scale_Min := -50.0;
   FP_PARM.Gradient_Time_ACC := 10;
   FP_PARM.AlarmLimit_H2 := 85.0;
   FP_PARM.AlarmLimit_H1 := 80.0;
   FP_PARM.AlarmDelay_H2_Pre := 5;
   FP_PARM.AlarmDelay_H2_Acc := 5;
   FP_PARM.AlarmDelay_H1_Pre := 5;
   FP_PARM.AlarmDelay_H1_Acc := 5;
   FP_PARM.OpenLoopDelay_Acc := 2;
   FP_PARM.OverRangeDelay_Acc := 2;
   ONS.SecPulse2 := TRUE;
   FIBUS_SubStatus := 16#FF;
   FIBUS_Quality := 16#FF;
   FIBUS_Limit := 16#FF;
   Result_Smooth := 45.74653;
   DampXEA := 45.74653;
   StatusWork := 1;
   AlarmDelay_H2_Mem := 5;
   AlarmDelay_H1_Mem := 5;
   GradientTime_Mem := 10;
   AlarmDelay_OpenLoop_Mem := 2;
   AlarmDelay_OverRange_Mem := 2;
   ScaledValue := 64.36632;
   Grad_OldValue := 64.36632;
   HystCalc := 2.5;
   OUT.PV_NORM := 45.74653;
   OUT.PV_SCAL := 64.36632;
   OUT.AL_H3 := TRUE;
   OUT.AL_H2 := TRUE;
   OUT.AL_H1 := TRUE;
   OUT.AL_L1 := TRUE;
   OUT.AL_L2 := TRUE;
   OUT.AL_L3 := TRUE;
   OUT.SIG_OK := TRUE;
   OUT.LIM_H2 := TRUE;
   OUT.LIM_H1 := TRUE;
   MSW_Status_Trans := 1;
END_DATA_BLOCK

DATA_BLOCK "_2010CR150A01T04_DB"   // DB5021
TITLE = Instance DB Analog: Temp
{ S7_Optimized_Access := 'FALSE' }
AUTHOR : METIS
NAME : ANA_DB
VERSION : 8.0
// stored: InstanceOfName ACESYS_ANALOG
"ACESYS_ANALOG"
BEGIN
   FP_EN.ParentSupress := TRUE;
   FP_EN.ParentSupressUnit := TRUE;
   FP_EN.Hysteresis := TRUE;
   FP_PARM.Scale_Max := 200.0;
   FP_PARM.Grad_Pos := 0.0;
   FP_PARM.Grad_Neg := 0.0;
   FP_PARM.OpenLoopDelay_Pre := 2;
   FP_PARM.Gradient_Time_Pre := 10;
   FP_PARM.Alarm_Hyst := 1.0;
   FP_PARM.OverRangeDelay_Pre := 2;
   FP_SIM.Value_Enable := TRUE;
   FP_SIM.Gain := 1.0;
   IN := 45.97078;
   U_RANGE := TRUE;
   O_RANGE := TRUE;
   SIG_FAULT := TRUE;
   EnConfig := TRUE;
   AEN := TRUE;
   PV_NORM := 45.97078;
   PV_SCAL := 64.92694;
   AL_H3 := TRUE;
   AL_H2 := TRUE;
   AL_H1 := TRUE;
   AL_L1 := TRUE;
   AL_L2 := TRUE;
   AL_L3 := TRUE;
   SIG_OK := TRUE;
   LIM_H2 := TRUE;
   LIM_H1 := TRUE;
   MSW.VALUE := 64.92694;
   MSW.TRIGVALUE := -67.70472;
   MSW.EXT.AlarmWarnUnAck := TRUE;
   MSW.EXT.Operation := TRUE;
   MSW.Status := 1;
   MSW.TimeStamp := 16#7303;
   BlockInfo.Ace_Version := 80;
   BlockInfo.Ace_BuildNo := 3;
   BlockInfo.DB_Number := 5021;
   FP_EN.Alarm_H2 := TRUE;
   FP_EN.Alarm_H1 := TRUE;
   FP_PARM.Scale_Min := -50.0;
   FP_PARM.Gradient_Time_ACC := 10;
   FP_PARM.AlarmLimit_H2 := 85.0;
   FP_PARM.AlarmLimit_H1 := 80.0;
   FP_PARM.AlarmDelay_H2_Pre := 5;
   FP_PARM.AlarmDelay_H2_Acc := 5;
   FP_PARM.AlarmDelay_H1_Pre := 5;
   FP_PARM.AlarmDelay_H1_Acc := 5;
   FP_PARM.OpenLoopDelay_Acc := 2;
   FP_PARM.OverRangeDelay_Acc := 2;
   ONS.SecPulse2 := TRUE;
   FIBUS_SubStatus := 16#FF;
   FIBUS_Quality := 16#FF;
   FIBUS_Limit := 16#FF;
   Result_Smooth := 45.97078;
   DampXEA := 45.97078;
   StatusWork := 1;
   AlarmDelay_H2_Mem := 5;
   AlarmDelay_H1_Mem := 5;
   GradientTime_Mem := 10;
   AlarmDelay_OpenLoop_Mem := 2;
   AlarmDelay_OverRange_Mem := 2;
   ScaledValue := 64.92694;
   Grad_OldValue := 64.92694;
   HystCalc := 2.5;
   OUT.PV_NORM := 45.97078;
   OUT.PV_SCAL := 64.92694;
   OUT.AL_H3 := TRUE;
   OUT.AL_H2 := TRUE;
   OUT.AL_H1 := TRUE;
   OUT.AL_L1 := TRUE;
   OUT.AL_L2 := TRUE;
   OUT.AL_L3 := TRUE;
   OUT.SIG_OK := TRUE;
   OUT.LIM_H2 := TRUE;
   OUT.LIM_H1 := TRUE;
   MSW_Status_Trans := 1;
END_DATA_BLOCK

DATA_BLOCK "_2010HP100L01_DB"   // DB5022
TITLE = Instance DB Analog: Level
{ S7_Optimized_Access := 'FALSE' }
AUTHOR : 7Art
NAME : ANA_DB
VERSION : 8.0
// stored: InstanceOfName ACESYS_ANALOG
"ACESYS_ANALOG"
BEGIN
   FP_EN.Hysteresis := TRUE;
   FP_PARM.Grad_Pos := 0.0;
   FP_PARM.Grad_Neg := 0.0;
   FP_PARM.OpenLoopDelay_Pre := 2;
   FP_PARM.Gradient_Time_Pre := 10;
   FP_PARM.Alarm_Hyst := 1.0;
   FP_PARM.OverRangeDelay_Pre := 2;
   FP_SIM.Value_Enable := TRUE;
   FP_SIM.Gain := 1.0;
   IN := 93.94893;
   U_RANGE := TRUE;
   O_RANGE := TRUE;
   SIG_FAULT := TRUE;
   EnConfig := TRUE;
   AEN := TRUE;
   PV_NORM := 93.94893;
   PV_SCAL := 93.94893;
   AL_H3 := TRUE;
   AL_H2 := TRUE;
   AL_H1 := TRUE;
   AL_L1 := TRUE;
   AL_L2 := TRUE;
   AL_L3 := TRUE;
   SIG_OK := TRUE;
   LIM_H2 := TRUE;
   LIM_H1 := TRUE;
   MSW.VALUE := 93.94893;
   MSW.TRIGVALUE := 94.01041;
   MSW.EXT.AlarmWarnUnAck := TRUE;
   MSW.EXT.Operation := TRUE;
   MSW.Status := 1;
   MSW.TimeStamp := 16#BAFA;
   BlockInfo.Ace_Version := 80;
   BlockInfo.Ace_BuildNo := 3;
   BlockInfo.DB_Number := 5022;
   FP_PARM.Gradient_Time_ACC := 10;
   FP_PARM.AlarmLimit_H2 := 85.0;
   FP_PARM.AlarmLimit_H1 := 80.0;
   FP_PARM.AlarmDelay_H2_Pre := 5;
   FP_PARM.AlarmDelay_H2_Acc := 5;
   FP_PARM.AlarmDelay_H1_Pre := 5;
   FP_PARM.AlarmDelay_H1_Acc := 5;
   FP_PARM.OpenLoopDelay_Acc := 2;
   FP_PARM.OverRangeDelay_Acc := 2;
   ONS.SecPulse2 := TRUE;
   FIBUS_SubStatus := 16#FF;
   FIBUS_Quality := 16#FF;
   FIBUS_Limit := 16#FF;
   Result_Smooth := 93.94893;
   DampXEA := 93.94893;
   StatusWork := 1;
   AlarmDelay_H2_Mem := 5;
   AlarmDelay_H1_Mem := 5;
   GradientTime_Mem := 10;
   AlarmDelay_OpenLoop_Mem := 2;
   AlarmDelay_OverRange_Mem := 2;
   ScaledValue := 93.94893;
   Grad_OldValue := 93.94893;
   HystCalc := 1.0;
   OUT.PV_NORM := 93.94893;
   OUT.PV_SCAL := 93.94893;
   OUT.AL_H3 := TRUE;
   OUT.AL_H2 := TRUE;
   OUT.AL_H1 := TRUE;
   OUT.AL_L1 := TRUE;
   OUT.AL_L2 := TRUE;
   OUT.AL_L3 := TRUE;
   OUT.SIG_OK := TRUE;
   OUT.LIM_H2 := TRUE;
   OUT.LIM_H1 := TRUE;
   MSW_Status_Trans := 1;
END_DATA_BLOCK

DATA_BLOCK "_2010CR150A01T05_DB"   // DB5023
TITLE = Instance DB Analog: Temp
{ S7_Optimized_Access := 'FALSE' }
AUTHOR : METIS
NAME : ANA_DB
VERSION : 8.0
// stored: InstanceOfName ACESYS_ANALOG
"ACESYS_ANALOG"
BEGIN
   FP_EN.ParentSupress := TRUE;
   FP_EN.ParentSupressUnit := TRUE;
   FP_EN.Hysteresis := TRUE;
   FP_PARM.Scale_Max := 80.0;
   FP_PARM.Grad_Pos := 0.0;
   FP_PARM.Grad_Neg := 0.0;
   FP_PARM.OpenLoopDelay_Pre := 2;
   FP_PARM.Gradient_Time_Pre := 10;
   FP_PARM.Alarm_Hyst := 1.0;
   FP_PARM.OverRangeDelay_Pre := 2;
   FP_SIM.Value_Enable := TRUE;
   FP_SIM.Gain := 1.0;
   IN := 45.72121;
   U_RANGE := TRUE;
   O_RANGE := TRUE;
   SIG_FAULT := TRUE;
   EnConfig := TRUE;
   AEN := TRUE;
   PV_NORM := 45.72121;
   PV_SCAL := 14.86546;
   AL_H3 := TRUE;
   AL_H2 := TRUE;
   AL_H1 := TRUE;
   AL_L1 := TRUE;
   AL_L2 := TRUE;
   AL_L3 := TRUE;
   SIG_OK := TRUE;
   LIM_H2 := TRUE;
   LIM_H1 := TRUE;
   MSW.VALUE := 14.86546;
   MSW.EXT.AlarmWarnUnAck := TRUE;
   MSW.EXT.Operation := TRUE;
   MSW.Status := 1;
   MSW.TimeStamp := 16#3928;
   BlockInfo.Ace_Version := 80;
   BlockInfo.Ace_BuildNo := 3;
   BlockInfo.DB_Number := 5023;
   FP_PARM.Scale_Min := -40.0;
   FP_PARM.Gradient_Time_ACC := 10;
   FP_PARM.AlarmLimit_H2 := 85.0;
   FP_PARM.AlarmLimit_H1 := 80.0;
   FP_PARM.AlarmDelay_H2_Pre := 5;
   FP_PARM.AlarmDelay_H2_Acc := 5;
   FP_PARM.AlarmDelay_H1_Pre := 5;
   FP_PARM.AlarmDelay_H1_Acc := 5;
   FP_PARM.OpenLoopDelay_Acc := 2;
   FP_PARM.OverRangeDelay_Acc := 2;
   ONS.SecPulse2 := TRUE;
   FIBUS_SubStatus := 16#FF;
   FIBUS_Quality := 16#FF;
   FIBUS_Limit := 16#FF;
   Result_Smooth := 45.72121;
   DampXEA := 45.72121;
   StatusWork := 1;
   AlarmDelay_H2_Mem := 5;
   AlarmDelay_H1_Mem := 5;
   GradientTime_Mem := 10;
   AlarmDelay_OpenLoop_Mem := 2;
   AlarmDelay_OverRange_Mem := 2;
   ScaledValue := 14.86546;
   Grad_OldValue := 14.86546;
   HystCalc := 1.2;
   OUT.PV_NORM := 45.72121;
   OUT.PV_SCAL := 14.86546;
   OUT.AL_H3 := TRUE;
   OUT.AL_H2 := TRUE;
   OUT.AL_H1 := TRUE;
   OUT.AL_L1 := TRUE;
   OUT.AL_L2 := TRUE;
   OUT.AL_L3 := TRUE;
   OUT.SIG_OK := TRUE;
   OUT.LIM_H2 := TRUE;
   OUT.LIM_H1 := TRUE;
   MSW_Status_Trans := 1;
END_DATA_BLOCK

DATA_BLOCK "_2010WG180N01F01_DB"   // DB5024
TITLE = Instance DB Analog: Weight Flow
{ S7_Optimized_Access := 'FALSE' }
AUTHOR : METIS
NAME : ANA_DB
VERSION : 8.0
// stored: InstanceOfName ACESYS_ANALOG
"ACESYS_ANALOG"
BEGIN
   FP_EN.ParentSupress := TRUE;
   FP_EN.ParentSupressUnit := TRUE;
   FP_EN.Hysteresis := TRUE;
   FP_PARM.Scale_Max := 1500.0;
   FP_PARM.Grad_Pos := 0.0;
   FP_PARM.Grad_Neg := 0.0;
   FP_PARM.OpenLoopDelay_Pre := 2;
   FP_PARM.Gradient_Time_Pre := 10;
   FP_PARM.Alarm_Hyst := 1.0;
   FP_PARM.OverRangeDelay_Pre := 2;
   FP_SIM.Value_Enable := TRUE;
   FP_SIM.Gain := 1.0;
   IN := -118.5185;
   U_RANGE := TRUE;
   O_RANGE := TRUE;
   SIG_FAULT := TRUE;
   EnConfig := TRUE;
   AEN := TRUE;
   AL_H3 := TRUE;
   AL_H2 := TRUE;
   AL_H1 := TRUE;
   AL_L1 := TRUE;
   AL_L2 := TRUE;
   AL_L3 := TRUE;
   SIG_OK := TRUE;
   LIM_H2 := TRUE;
   LIM_H1 := TRUE;
   LIM_L1 := TRUE;
   LIM_L2 := TRUE;
   MSW.EXT.AlarmWarnUnAck := TRUE;
   MSW.EXT.Operation := TRUE;
   MSW.EXT.Forced := TRUE;
   MSW.Status := 1;
   MSW.TimeStamp := 16#3928;
   BlockInfo.Ace_Version := 80;
   BlockInfo.Ace_BuildNo := 3;
   BlockInfo.DB_Number := 5024;
   FP_EN.Force := TRUE;
   FP_PARM.Gradient_Time_ACC := 10;
   FP_PARM.AlarmLimit_H2 := 85.0;
   FP_PARM.AlarmLimit_H1 := 80.0;
   FP_PARM.AlarmDelay_H2_Pre := 5;
   FP_PARM.AlarmDelay_H2_Acc := 5;
   FP_PARM.AlarmDelay_H1_Pre := 5;
   FP_PARM.AlarmDelay_H1_Acc := 5;
   FP_PARM.OpenLoopDelay_Acc := 2;
   FP_PARM.OverRangeDelay_Acc := 2;
   ONS.SecPulse2 := TRUE;
   FIBUS_SubStatus := 16#FF;
   FIBUS_Quality := 16#FF;
   FIBUS_Limit := 16#FF;
   StatusWork := 1;
   AlarmDelay_H2_Mem := 5;
   AlarmDelay_H1_Mem := 5;
   GradientTime_Mem := 10;
   AlarmDelay_OpenLoop_Mem := 2;
   AlarmDelay_OverRange_Mem := 2;
   HystCalc := 15.0;
   OUT.AL_H3 := TRUE;
   OUT.AL_H2 := TRUE;
   OUT.AL_H1 := TRUE;
   OUT.AL_L1 := TRUE;
   OUT.AL_L2 := TRUE;
   OUT.AL_L3 := TRUE;
   OUT.SIG_OK := TRUE;
   OUT.LIM_H2 := TRUE;
   OUT.LIM_H1 := TRUE;
   OUT.LIM_L1 := TRUE;
   OUT.LIM_L2 := TRUE;
   MSW_Status_Trans := 1;
END_DATA_BLOCK

DATA_BLOCK "_2010PMC01A01T01_DB"   // DB5025
{ S7_Optimized_Access := 'FALSE' }
AUTHOR : FLSmidth
FAMILY : ACESYS
NAME : ANALOG
VERSION : 8.0
// stored: InstanceOfName ACESYS_ANALOG
"ACESYS_ANALOG"
BEGIN
END_DATA_BLOCK

DATA_BLOCK "_2015SU026N01L01_DB"   // DB5476
TITLE = Instance DB Analog:
{ S7_Optimized_Access := 'FALSE' }
AUTHOR : METIS
NAME : ANA_DB
VERSION : 8.0
// stored: InstanceOfName ACESYS_ANALOG
"ACESYS_ANALOG"
BEGIN
   FP_EN.ParentSupress := TRUE;
   FP_EN.ParentSupressUnit := TRUE;
   FP_PARM.Grad_Pos := 0.0;
   FP_PARM.Grad_Neg := 0.0;
   FP_PARM.Gradient_Time_Pre := 10;
   FP_SIM.Gain := 1.0;
   FP_SIM.Value_Enable := TRUE;
   IN := -0.03255208;
   U_RANGE := TRUE;
   O_RANGE := TRUE;
   SIG_FAULT := TRUE;
   EnConfig := TRUE;
   AEN := TRUE;
   AL_SUPR := TRUE;
   PV_NORM := -0.03255208;
   PV_SCAL := -0.03255208;
   AL_H3 := TRUE;
   AL_H2 := TRUE;
   AL_H1 := TRUE;
   AL_L1 := TRUE;
   AL_L2 := TRUE;
   AL_L3 := TRUE;
   SIG_OK := TRUE;
   LIM_L1 := TRUE;
   LIM_L2 := TRUE;
   MSW.VALUE := -0.03255208;
   MSW.TRIGVALUE := 108.878;
   MSW.EXT.AlarmWarnUnAck := TRUE;
   MSW.EXT.Operation := TRUE;
   MSW.EXT.AlarmSuppressed := TRUE;
   MSW.Status := 1;
   MSW.TimeStamp := 16#9A3E;
   BlockInfo.Ace_Version := 80;
   BlockInfo.Ace_BuildNo := 3;
   BlockInfo.DB_Number := 5476;
   FP_EN.Alarm_H2 := TRUE;
   FP_EN.AlarmDelay_H2 := TRUE;
   FP_PARM.Gradient_Time_ACC := 10;
   FP_PARM.AlarmLimit_H2 := 110.0;
   FP_PARM.AlarmDelay_H2_Pre := 3;
   FP_PARM.AlarmDelay_H2_Acc := 3;
   ONS.SecPulse2 := TRUE;
   FIBUS_SubStatus := 16#FF;
   FIBUS_Quality := 16#FF;
   FIBUS_Limit := 16#FF;
   Result_Smooth := -0.03255208;
   DampXEA := -0.03255208;
   ALARM_SuppresionActiv := TRUE;
   StatusWork := 1;
   AlarmDelay_H2_Mem := 3;
   GradientTime_Mem := 10;
   ScaledValue := -0.03255208;
   Grad_OldValue := -0.03255208;
   OUT.PV_NORM := -0.03255208;
   OUT.PV_SCAL := -0.03255208;
   OUT.AL_H3 := TRUE;
   OUT.AL_H2 := TRUE;
   OUT.AL_H1 := TRUE;
   OUT.AL_L1 := TRUE;
   OUT.AL_L2 := TRUE;
   OUT.AL_L3 := TRUE;
   OUT.SIG_OK := TRUE;
   OUT.LIM_L1 := TRUE;
   OUT.LIM_L2 := TRUE;
   MSW_Status_Trans := 1;
END_DATA_BLOCK

DATA_BLOCK "_2015PU027N01F01_DB"   // DB5478
TITLE = Instance DB Analog:
{ S7_Optimized_Access := 'FALSE' }
AUTHOR : METIS
NAME : ANA_DB
VERSION : 8.0
// stored: InstanceOfName ACESYS_ANALOG
"ACESYS_ANALOG"
BEGIN
   FP_EN.ParentSupress := TRUE;
   FP_EN.ParentSupressUnit := TRUE;
   FP_PARM.Grad_Pos := 0.0;
   FP_PARM.Grad_Neg := 0.0;
   FP_PARM.Gradient_Time_Pre := 10;
   FP_SIM.Gain := 1.0;
   FP_SIM.Value_Enable := TRUE;
   IN := 40.99031;
   U_RANGE := TRUE;
   O_RANGE := TRUE;
   SIG_FAULT := TRUE;
   EnConfig := TRUE;
   AEN := TRUE;
   AL_SUPR := TRUE;
   PV_NORM := 40.99031;
   PV_SCAL := 40.99031;
   AL_H3 := TRUE;
   AL_H2 := TRUE;
   AL_H1 := TRUE;
   AL_L1 := TRUE;
   AL_L2 := TRUE;
   AL_L3 := TRUE;
   SIG_OK := TRUE;
   LIM_H2 := TRUE;
   LIM_H1 := TRUE;
   MSW.VALUE := 40.99031;
   MSW.EXT.AlarmWarnUnAck := TRUE;
   MSW.EXT.Operation := TRUE;
   MSW.EXT.AlarmSuppressed := TRUE;
   MSW.Status := 1;
   MSW.TimeStamp := 16#08C9;
   BlockInfo.Ace_Version := 80;
   BlockInfo.Ace_BuildNo := 3;
   BlockInfo.DB_Number := 5478;
   FP_PARM.Gradient_Time_ACC := 10;
   ONS.SecPulse2 := TRUE;
   FIBUS_SubStatus := 16#FF;
   FIBUS_Quality := 16#FF;
   FIBUS_Limit := 16#FF;
   Result_Smooth := 40.99031;
   DampXEA := 40.99031;
   ALARM_SuppresionActiv := TRUE;
   StatusWork := 1;
   GradientTime_Mem := 10;
   ScaledValue := 40.99031;
   Grad_OldValue := 40.99031;
   OUT.PV_NORM := 40.99031;
   OUT.PV_SCAL := 40.99031;
   OUT.AL_H3 := TRUE;
   OUT.AL_H2 := TRUE;
   OUT.AL_H1 := TRUE;
   OUT.AL_L1 := TRUE;
   OUT.AL_L2 := TRUE;
   OUT.AL_L3 := TRUE;
   OUT.SIG_OK := TRUE;
   OUT.LIM_H2 := TRUE;
   OUT.LIM_H1 := TRUE;
   MSW_Status_Trans := 1;
END_DATA_BLOCK

DATA_BLOCK "_2015SU026N02F01_DB"   // DB5479
TITLE = Instance DB Analog:
{ S7_Optimized_Access := 'FALSE' }
AUTHOR : METIS
NAME : ANA_DB
VERSION : 8.0
// stored: InstanceOfName ACESYS_ANALOG
"ACESYS_ANALOG"
BEGIN
   FP_EN.ParentSupress := TRUE;
   FP_EN.ParentSupressUnit := TRUE;
   FP_PARM.Grad_Pos := 0.0;
   FP_PARM.Grad_Neg := 0.0;
   FP_PARM.Gradient_Time_Pre := 10;
   FP_SIM.Gain := 1.0;
   FP_SIM.Value_Enable := TRUE;
   IN := 0.03255208;
   U_RANGE := TRUE;
   O_RANGE := TRUE;
   SIG_FAULT := TRUE;
   EnConfig := TRUE;
   AEN := TRUE;
   AL_SUPR := TRUE;
   PV_NORM := 0.03255208;
   PV_SCAL := 0.03255208;
   AL_H3 := TRUE;
   AL_H2 := TRUE;
   AL_H1 := TRUE;
   AL_L1 := TRUE;
   AL_L2 := TRUE;
   AL_L3 := TRUE;
   SIG_OK := TRUE;
   LIM_H2 := TRUE;
   LIM_H1 := TRUE;
   MSW.VALUE := 0.03255208;
   MSW.EXT.AlarmWarnUnAck := TRUE;
   MSW.EXT.Operation := TRUE;
   MSW.EXT.AlarmSuppressed := TRUE;
   MSW.Status := 1;
   MSW.TimeStamp := 16#08C9;
   BlockInfo.Ace_Version := 80;
   BlockInfo.Ace_BuildNo := 3;
   BlockInfo.DB_Number := 5479;
   FP_PARM.Gradient_Time_ACC := 10;
   ONS.SecPulse2 := TRUE;
   FIBUS_SubStatus := 16#FF;
   FIBUS_Quality := 16#FF;
   FIBUS_Limit := 16#FF;
   Result_Smooth := 0.03255208;
   DampXEA := 0.03255208;
   ALARM_SuppresionActiv := TRUE;
   StatusWork := 1;
   GradientTime_Mem := 10;
   ScaledValue := 0.03255208;
   Grad_OldValue := 0.03255208;
   OUT.PV_NORM := 0.03255208;
   OUT.PV_SCAL := 0.03255208;
   OUT.AL_H3 := TRUE;
   OUT.AL_H2 := TRUE;
   OUT.AL_H1 := TRUE;
   OUT.AL_L1 := TRUE;
   OUT.AL_L2 := TRUE;
   OUT.AL_L3 := TRUE;
   OUT.SIG_OK := TRUE;
   OUT.LIM_H2 := TRUE;
   OUT.LIM_H1 := TRUE;
   MSW_Status_Trans := 1;
END_DATA_BLOCK

DATA_BLOCK "_2015SU026I01_DB"   // DB6054
TITLE = Instance DB PID:
{ S7_Optimized_Access := 'FALSE' }
AUTHOR : METIS
NAME : PID_DB
VERSION : 8.0
// stored: InstanceOfName ACESYS_PID
"ACESYS_PID"
BEGIN
   FP_EN.HLC_Track := TRUE;
   FP_PARM.DevFault_Limit := 100.0;
   FP_PARM.DevFault_Time_PRE := 60;
   PV := -0.03255208;
   PV_OK := TRUE;
   INV := TRUE;
   CYCLE := 100;
   SPNORM := 10.0;
   AUTO := TRUE;
   MSW.EXT.Operation := TRUE;
   MSW.Status := 1;
   MSW.TimeStamp := 16#1FD1;
   SPA := 10.0;
   SPA_HLC := 10.0;
   BlockInfo.Ace_Version := 80;
   BlockInfo.Ace_BuildNo := 3;
   BlockInfo.State_Act := 50;
   BlockInfo.State_Prev := 52;
   BlockInfo.DB_Number := 6054;
   FP_CMD.Auto := TRUE;
   FP_CMD.Internal := TRUE;
   FP_DIM.Manual := TRUE;
   FP_DIM.LastSP := TRUE;
   FP_DIM.AutoTune_Start_TIR := TRUE;
   FP_DIM.AutoTune_Ack := TRUE;
   FP_DIM.AutoTune_Undo := TRUE;
   FP_DIM.AutoTune_Start_SUT := TRUE;
   FP_SHOW.PB_Manual := TRUE;
   FP_SHOW.PB_Auto := TRUE;
   FP_SHOW.PB_LastSP := TRUE;
   FP_PARM.OUT_Max_Lim := 67.0;
   FP_PARM.LastSPA := 20.0;
   FP_PARM.DeadBand_High := 0.0;
   FP_PARM.DeadBand_Low := 0.0;
   FP_PARM.DevFault_Time_ACC := 60;
   FP_PARM_TIA.AutoTune_TIR_Phase := 1;
   FP_PARM_TIA.AutoTune_TIA_FP := 100;
   FP_PARM_TIA.AutoTune_SUT_TuneRule_0 := TRUE;
   FP_PARM_TIA.AutoTune_TIR_TuneRule_0 := TRUE;
   FP_PARM_TIA.WarningBit05 := TRUE;
   STATE.AUTO_Int := TRUE;
   ONS.FP_Auto1 := TRUE;
   ONS.FP_Auto2 := TRUE;
   ONS.FP_Int := TRUE;
   ONS.SecPulse2 := TRUE;
   ONS.Self_Auto := TRUE;
   ONS.SUT_TuneRule_0 := TRUE;
   ONS.TIR_TuneRule_0 := TRUE;
   OutDB_Low := TRUE;
   From_Pid_ErrorBits := 16#0000_0000;
   DevFault_Time_Men := 60;
   StatusWork := 1;
   DI_PID.Setpoint := 10.0;
   DI_PID.State := 3;
   DI_PID.ErrorBits := 16#0000_0000;
   DI_PID.Mode := 3;
   MSW_Status := 1;
END_DATA_BLOCK

DATA_BLOCK "_2010CV180N01Q41_DB"   // DB7000
TITLE = Instance DB Totalizer: _2010WG038N01Q41
{ S7_Optimized_Access := 'FALSE' }
AUTHOR : METIS
NAME : COUNT_DB
VERSION : 8.0
// stored: InstanceOfName ACESYS_TOTALIZER
"ACESYS_TOTALIZER"
BEGIN
   FP_EN.Reset := TRUE;
   FP_SEL.AI_Type_3 := TRUE;
   FP_SEL.COUNT_Factor_1 := TRUE;
   CNT_EN := TRUE;
   RESET := TRUE;
   COUNT := 1.0;
   MSW := 1;
   BlockInfo.Ace_Version := 80;
   BlockInfo.Ace_BuildNo := 3;
   BlockInfo.DB_Number := 7000;
   FP_SEL.User_Defined := TRUE;
   FP_PAR.Prev_Year := 1.0;
   FP_DIM.Reset := TRUE;
   FP_SHOW.Reset := TRUE;
   ONS.AI_Type_3 := TRUE;
   ONS.COUNT_Factor_1 := TRUE;
   ONS.User_Defined := TRUE;
   ONS.Reset := TRUE;
   ONS.SecPulse1 := TRUE;
   inc_tmr_Real := 26.3034;
   Selected_Factor := 1.0;
   User_int := 1.0;
   Runtime_Result := 0.0263034;
   Runtime_Mem1 := 16#0000_A80C_A687_D0A6;
END_DATA_BLOCK

DATA_BLOCK "_2010CV120M01_MAINT"   // DB8000
{ S7_Optimized_Access := 'FALSE' }
VERSION : 0.1
// stored: InstanceOfName Eqip_Maintenance
"Eqip_Maintenance"
BEGIN
   IN := TRUE;
   Cnt_Hours_1 := 5554;
   Cnt_Hours_2 := 6246;
   Cnt_Hours_3 := 6246;
   Cnt_Hours_4 := 6246;
   Accum_1 := 19994965;
   Accum_2 := 22486585;
   Accum_3 := 22486585;
   Accum_4 := 22486585;
END_DATA_BLOCK

DATA_BLOCK "_2010CV180U01_MAINT"   // DB8001
{ S7_Optimized_Access := 'FALSE' }
VERSION : 0.1
// stored: InstanceOfName Eqip_Maintenance
"Eqip_Maintenance"
BEGIN
   IN := TRUE;
   Cnt_Hours_1 := 4598;
   Cnt_Hours_2 := 6305;
   Cnt_Hours_3 := 6305;
   Cnt_Hours_4 := 6305;
   Accum_1 := 16556150;
   Accum_2 := 22698735;
   Accum_3 := 22698735;
   Accum_4 := 22698735;
END_DATA_BLOCK

DATA_BLOCK "_2010CV300U01_MAINT"   // DB8002
{ S7_Optimized_Access := 'FALSE' }
VERSION : 0.1
// stored: InstanceOfName Eqip_Maintenance
"Eqip_Maintenance"
BEGIN
   Accum_1 := 18862160;
   IN := TRUE;
   Cnt_Hours_1 := 5239;
   Cnt_Hours_2 := 6307;
   Cnt_Hours_3 := 6307;
   Cnt_Hours_4 := 6307;
   Accum_2 := 22708080;
   Accum_3 := 22708080;
   Accum_4 := 22708080;
END_DATA_BLOCK

DATA_BLOCK "_2010SC130U01_MAINT"   // DB8003
{ S7_Optimized_Access := 'FALSE' }
VERSION : 0.1
// stored: InstanceOfName Eqip_Maintenance
"Eqip_Maintenance"
BEGIN
   Accum_1 := 1189075;
   IN := TRUE;
   Cnt_Hours_1 := 330;
   Cnt_Hours_2 := 6202;
   Cnt_Hours_3 := 6202;
   Cnt_Hours_4 := 6202;
   Accum_2 := 22329700;
   Accum_3 := 22329700;
   Accum_4 := 22329700;
END_DATA_BLOCK

DATA_BLOCK "_2010BF110U01_MAINT"   // DB8004
{ S7_Optimized_Access := 'FALSE' }
VERSION : 0.1
// stored: InstanceOfName Eqip_Maintenance
"Eqip_Maintenance"
BEGIN
   Accum_1 := 18237740;
   IN := TRUE;
   Cnt_Hours_1 := 5066;
   Cnt_Hours_2 := 6113;
   Cnt_Hours_3 := 6113;
   Cnt_Hours_4 := 6113;
   Accum_2 := 22007375;
   Accum_3 := 22007375;
   Accum_4 := 22007375;
END_DATA_BLOCK

DATA_BLOCK "_2010CR150M01_MAINT"   // DB8005
{ S7_Optimized_Access := 'FALSE' }
VERSION : 0.1
// stored: InstanceOfName Eqip_Maintenance
"Eqip_Maintenance"
BEGIN
   Accum_1 := 1218045;
   IN := TRUE;
   Cnt_Hours_1 := 338;
   Cnt_Hours_2 := 6302;
   Cnt_Hours_3 := 6302;
   Cnt_Hours_4 := 6302;
   Accum_2 := 22690265;
   Accum_3 := 22690265;
   Accum_4 := 22690265;
END_DATA_BLOCK

DATA_BLOCK "_2010OB190M01_MAINT"   // DB8007
{ S7_Optimized_Access := 'FALSE' }
VERSION : 0.1
// stored: InstanceOfName Eqip_Maintenance
"Eqip_Maintenance"
BEGIN
   IN := TRUE;
   Cnt_Hours_1 := 1341;
   Cnt_Hours_2 := 1341;
   Cnt_Hours_3 := 1341;
   Cnt_Hours_4 := 1341;
   Accum_1 := 4828135;
   Accum_2 := 4828135;
   Accum_3 := 4828135;
   Accum_4 := 4828135;
END_DATA_BLOCK

DATA_BLOCK "2015PU035U01_MAINT"   // DB8009
{ S7_Optimized_Access := 'FALSE' }
VERSION : 0.1
// stored: InstanceOfName Eqip_Maintenance
"Eqip_Maintenance"
BEGIN
   Cnt_Hours_1 := 237;
   Cnt_Hours_2 := 237;
   Cnt_Hours_3 := 237;
   Cnt_Hours_4 := 237;
   Accum_1 := 855360;
   Accum_2 := 855360;
   Accum_3 := 855360;
   Accum_4 := 855360;
END_DATA_BLOCK

DATA_BLOCK "2015PU027U01_MAINT"   // DB8010
{ S7_Optimized_Access := 'FALSE' }
VERSION : 0.1
// stored: InstanceOfName Eqip_Maintenance
"Eqip_Maintenance"
BEGIN
   Cnt_Hours_1 := 535;
   Cnt_Hours_2 := 535;
   Cnt_Hours_3 := 535;
   Cnt_Hours_4 := 535;
   Accum_1 := 1928480;
   Accum_2 := 1928480;
   Accum_3 := 1928480;
   Accum_4 := 1928480;
END_DATA_BLOCK

DATA_BLOCK "2015PU028U01_MAINT"   // DB8011
{ S7_Optimized_Access := 'FALSE' }
VERSION : 0.1
// stored: InstanceOfName Eqip_Maintenance
"Eqip_Maintenance"
BEGIN
   Cnt_Hours_2 := 700;
   Cnt_Hours_3 := 700;
   Cnt_Hours_4 := 700;
   Accum_1 := 665;
   Accum_2 := 2523390;
   Accum_3 := 2523390;
   Accum_4 := 2523390;
END_DATA_BLOCK

DATA_BLOCK "2015PU040M01_MAINT"   // DB8012
{ S7_Optimized_Access := 'FALSE' }
VERSION : 0.1
// stored: InstanceOfName Eqip_Maintenance
"Eqip_Maintenance"
BEGIN
   IN := TRUE;
   Cnt_Hours_1 := 2963;
   Cnt_Hours_2 := 2963;
   Cnt_Hours_3 := 2963;
   Cnt_Hours_4 := 2963;
   Accum_1 := 10670300;
   Accum_2 := 10670300;
   Accum_3 := 10670300;
   Accum_4 := 10670300;
END_DATA_BLOCK

DATA_BLOCK "2015PU041M01_MAINT"   // DB8013
{ S7_Optimized_Access := 'FALSE' }
VERSION : 0.1
// stored: InstanceOfName Eqip_Maintenance
"Eqip_Maintenance"
BEGIN
   Cnt_Hours_1 := 1762;
   Cnt_Hours_2 := 1762;
   Cnt_Hours_3 := 1762;
   Cnt_Hours_4 := 1762;
   Accum_1 := 6344850;
   Accum_2 := 6344845;
   Accum_3 := 6344840;
   Accum_4 := 6344835;
END_DATA_BLOCK

DATA_BLOCK "2015PU042M01_MAINT"   // DB8014
{ S7_Optimized_Access := 'FALSE' }
VERSION : 0.1
// stored: InstanceOfName Eqip_Maintenance
"Eqip_Maintenance"
BEGIN
   IN := TRUE;
   Cnt_Hours_1 := 4845;
   Cnt_Hours_2 := 4845;
   Cnt_Hours_3 := 4845;
   Cnt_Hours_4 := 4845;
   Accum_1 := 17443825;
   Accum_2 := 17443825;
   Accum_3 := 17443825;
   Accum_4 := 17443825;
END_DATA_BLOCK

DATA_BLOCK "TX05_RX04_01"   // DB10000
{ S7_Optimized_Access := 'TRUE' }
VERSION : 0.1
// stored: InstanceOfName ACESYS_SEND
"ACESYS_SEND"
BEGIN
   Primary_EN := TRUE;
   Primary_ID := 16#00C1;
   Primary_DEV_ID := 16#10;
   Primary_ACT := TRUE;
   Primary_IP_ADDR1 := 10;
   Primary_IP_ADDR2 := 26;
   Primary_IP_ADDR3 := 206;
   Primary_IP_ADDR4 := 11;
   Primary_LOC_RS := 16#02;
   Primary_CP_RS := 16#02;
   Primary_REM_RS := 16#02;
   Secondary_ID := 16#00C2;
   Secondary_ACT := TRUE;
   Secondary_LOC_RS := 16#02;
   Secondary_REM_RS := 16#02;
   DATA.BOOLEAN[5] := TRUE;
   DATA.BOOLEAN[6] := TRUE;
   DATA.REAL_VAL[0] := 67.37196;
   MASTER_LINK.Flash_Slow := TRUE;
   MASTER_LINK.Flash_Fast := TRUE;
   MASTER_LINK.SS_FP_Enable := TRUE;
   MASTER_LINK.Man_Enable := TRUE;
   MASTER_LINK.Loc_Enable := TRUE;
   MASTER_LINK.Test_Enable := TRUE;
   MASTER_LINK.TimeStamp := 16#6BEB;
   MASTER_LINK.OB1_CycleTime := 2;
   Primary_Comm_OK := TRUE;
   Primary_Conn_St := 16#80C4;
   Primary_Send_St := 16#7000;
   Secondary_Send_St := 16#7000;
   BlockInfo.Ace_Version := 80;
   BlockInfo.Ace_BuildNo := 3;
   BlockInfo.DB_Number := 10000;
   PRIM_T_SEND.ID := 16#00C1;
   PRIM_T_SEND.LEN := 106;
   PRIM_T_SEND.STATUS := 16#7000;
   PRIM_T_CONN.REQ := TRUE;
   PRIM_T_CONN.ID := 16#00C1;
   PRIM_T_CONN.DONE := TRUE;
   PRIM_T_DISC.ID := 16#00C1;
   PRIM_T_DISC.STATUS := 16#7000;
   PRIM_T_PARAM.InterfaceId := 259;
   PRIM_T_PARAM.ID := 16#00C1;
   PRIM_T_PARAM.ConnectionType := 16#0C;
   PRIM_T_PARAM.ActiveEstablished := TRUE;
   PRIM_T_PARAM.RemoteAddress.ADDR[1] := 16#0A;
   PRIM_T_PARAM.RemoteAddress.ADDR[2] := 16#1A;
   PRIM_T_PARAM.RemoteAddress.ADDR[3] := 16#CE;
   PRIM_T_PARAM.RemoteAddress.ADDR[4] := 16#0B;
   PRIM_T_PARAM.RemoteTSelector.TSelLength := 6;
   PRIM_T_PARAM.RemoteTSelector.TSel[1] := 16#E0;
   PRIM_T_PARAM.RemoteTSelector.TSel[2] := 16#02;
   PRIM_T_PARAM.RemoteTSelector.TSel[3] := 16#2B;
   PRIM_T_PARAM.RemoteTSelector.TSel[4] := 16#31;
   PRIM_T_PARAM.RemoteTSelector.TSel[5] := 16#39;
   PRIM_T_PARAM.RemoteTSelector.TSel[6] := 16#33;
   PRIM_T_PARAM.LocalTSelector.TSelLength := 6;
   PRIM_T_PARAM.LocalTSelector.TSel[1] := 16#E0;
   PRIM_T_PARAM.LocalTSelector.TSel[2] := 16#02;
   PRIM_T_PARAM.LocalTSelector.TSel[3] := 16#2B;
   PRIM_T_PARAM.LocalTSelector.TSel[4] := 16#31;
   PRIM_T_PARAM.LocalTSelector.TSel[5] := 16#39;
   PRIM_T_PARAM.LocalTSelector.TSel[6] := 16#33;
   PRIM_CONN_DATA.REGISTERED := TRUE;
   PRIM_CONN_DATA.CONN_DONE := TRUE;
   PRIM_CONN_DATA.STATUS_SAV := -32572;
   PRIM_CONN_DATA.SEND_REQ_I := TRUE;
   PRIM_CONN_DATA.SEND_STATUS := 16#7000;
   PRIM_CONN_DATA.ABORT_STATUS := 16#7000;
   SEC_T_SEND.ID := 16#00C2;
   SEC_T_SEND.LEN := 106;
   SEC_T_SEND.STATUS := 16#7000;
   SEC_T_CONN.STATUS := 16#7000;
   SEC_T_DISC.REQ := TRUE;
   SEC_T_DISC.ID := 16#00C2;
   SEC_T_DISC.STATUS := 16#7000;
   SEC_T_PARAM.ID := 16#00C2;
   SEC_T_PARAM.ConnectionType := 16#0C;
   SEC_T_PARAM.ActiveEstablished := TRUE;
   SEC_T_PARAM.RemoteTSelector.TSelLength := 6;
   SEC_T_PARAM.RemoteTSelector.TSel[1] := 16#E0;
   SEC_T_PARAM.RemoteTSelector.TSel[2] := 16#02;
   SEC_T_PARAM.RemoteTSelector.TSel[3] := 16#2B;
   SEC_T_PARAM.RemoteTSelector.TSel[4] := 16#31;
   SEC_T_PARAM.RemoteTSelector.TSel[5] := 16#39;
   SEC_T_PARAM.RemoteTSelector.TSel[6] := 16#34;
   SEC_T_PARAM.LocalTSelector.TSelLength := 6;
   SEC_T_PARAM.LocalTSelector.TSel[1] := 16#E0;
   SEC_T_PARAM.LocalTSelector.TSel[2] := 16#02;
   SEC_T_PARAM.LocalTSelector.TSel[3] := 16#2B;
   SEC_T_PARAM.LocalTSelector.TSel[4] := 16#31;
   SEC_T_PARAM.LocalTSelector.TSel[5] := 16#39;
   SEC_T_PARAM.LocalTSelector.TSel[6] := 16#34;
   SEC_CONN_DATA.REGISTERED := TRUE;
   SEC_CONN_DATA.SEND_REQ_P := TRUE;
   SEC_CONN_DATA.SEND_STATUS := 16#7000;
   SEC_CONN_DATA.ABORT_REQ := TRUE;
   SEC_CONN_DATA.ABORT_REQ_I := TRUE;
   SEC_CONN_DATA.ABORT_REQ_P := TRUE;
   SEC_CONN_DATA.ABORT_STATUS := 16#7000;
   TSAP16 := '+194';
   Prim_String := '+193';
   Sec_String := '+194';
   Prim_En_ONS := TRUE;
   Prim_SendReq_Dn := TRUE;
   Prim_EN := TRUE;
   Primary_ID_Old := 16#00C1;
   Secondary_ID_Old := 16#00C2;
   Prim_Con_TMR.ST := T#-22D_23H_2M_59S_467MS;
   Prim_Con_TMR.PT := T#4S;
   Prim_Del_ReCon.ST := T#21D_3H_22M_43S_545MS;
   Prim_Del_ReCon.PT := T#7S;
   Sec_Del_ReCon.ST := T#-6D_22H_42M_42S_994MS;
   Sec_Del_ReCon.PT := T#5S;
   Prim_Com_OK.ST := T#20D_14H_53M_47S_254MS;
   Prim_Com_OK.PT := T#1S;
   Prim_Com_OK.IN := TRUE;
   Prim_SendDelay.ST := T#21D_3H_22M_43S_551MS;
   Prim_SendDelay.PT := T#400MS;
   Prim_SendDelay.RU := TRUE;
   Prim_SendDelay.IN := TRUE;
   PRIM_EXT_HWID.HWTYPE := 4;
   PRIM_EXT_HWID.SLOT := 2;
   SEC_EXT_HWID.HWTYPE := 4;
END_DATA_BLOCK

DATA_BLOCK "_2010CV300U01_AD"   // DB14007
{ S7_Optimized_Access := 'FALSE' }
VERSION : 0.1
// stored: InstanceOfName IUSYS_INVT_PN_MOTOR
"IUSYS_INVT_PN_MOTOR"
BEGIN
   INREF := 500;
   OUTREF := 500;
   FUNCTYPE := 41;
   NET := 101;
   NODE := 3;
   CV := 110.0;
   MCC := TRUE;
   RDY := TRUE;
   OVL := TRUE;
   RET1 := TRUE;
   LSTP := TRUE;
   REM := TRUE;
   SSW := TRUE;
   TFA := TRUE;
   DRDY := TRUE;
   STALL := TRUE;
   EARTH := TRUE;
   UBAL := TRUE;
   GFA := TRUE;
   GWA := TRUE;
   BUSF := TRUE;
   DOPR := TRUE;
   AI1 := 243.2;
   AI2 := 55.1;
   AI3 := 110.86;
   RAW_Input.SB00_0 := TRUE;
   RAW_Input.SB00_6 := TRUE;
   RAW_Input.SB01 := 16#02;
   RAW_Input.SW02 := 16#15A7;
   RAW_Input.SW04 := 551;
   RAW_Input.SW08 := 2432;
   RAW_Input.SW22 := 16#FE81;
   RAW_Output.CB01 := 16#01;
   RAW_Output.CW02 := 16#157C;
   RAW_Output.CW08 := 16#0001;
   IHK.DelSTR_Timer_PV := 1;
   IHK.DelSTP_Timer_PV := 3;
   IHK.DelSTP_Timer_Mem := 3;
   IHK.RES_Timer_PV := 2;
   IHK.RES_Timer_Mem := 2;
   IHK.ChgOverTime_PV := 1;
   IHK.ChgOverTime_Mem := 1;
   IHK.CoastTimer_PV := 1;
   IHK.CoastTimer_Mem := 1;
   IHK.DelSTR_Timer_DN := TRUE;
   IHK.AUX_DelSTR_Time := 1;
   IHK.CoastSTP := TRUE;
   IHK.ComON := TRUE;
   IHK.Aux_CB01_0 := TRUE;
   IHK.No_Acyc := TRUE;
   IHK.Pulse._01 := TRUE;
   IHK.Pulse._03 := TRUE;
   AC.Ons_Read_Req := TRUE;
   AC.Motor_Data_99._06 := 100.0;
   AC.Motor_Data_99._09 := 100;
   AC.Motor_Data_99._10 := 100.0;
   AC._99_Status := 16#0000_0000;
   AC_Read_99_Migra.STATUS := 16#0000_0000;
   OUT.MCC := TRUE;
   OUT.RDY := TRUE;
   OUT.OVL := TRUE;
   OUT.RET1 := TRUE;
   OUT.LSTP := TRUE;
   OUT.REM := TRUE;
   OUT.SSW := TRUE;
   OUT.TFA := TRUE;
   OUT.DRDY := TRUE;
   OUT.STALL := TRUE;
   OUT.EARTH := TRUE;
   OUT.UBAL := TRUE;
   OUT.GFA := TRUE;
   OUT.GWA := TRUE;
   OUT.BUSF := TRUE;
   OUT.DOPR := TRUE;
   OUT.AI1 := 243.2;
   OUT.AI2 := 55.1;
   OUT.AI3 := 110.86;
END_DATA_BLOCK

DATA_BLOCK "_2010CV180U01_AD"   // DB14008
{ S7_Optimized_Access := 'FALSE' }
VERSION : 0.1
// stored: InstanceOfName IUSYS_INVT_PN_MOTOR
"IUSYS_INVT_PN_MOTOR"
BEGIN
   INREF := 532;
   OUTREF := 532;
   FUNCTYPE := 41;
   NET := 101;
   NODE := 3;
   CV := 90.0;
   MCC := TRUE;
   RDY := TRUE;
   OVL := TRUE;
   RET1 := TRUE;
   LSTP := TRUE;
   REM := TRUE;
   SSW := TRUE;
   TFA := TRUE;
   DRDY := TRUE;
   STALL := TRUE;
   EARTH := TRUE;
   UBAL := TRUE;
   GFA := TRUE;
   GWA := TRUE;
   BUSF := TRUE;
   DOPR := TRUE;
   AI1 := 62.9;
   AI2 := 29.2;
   AI3 := 90.0;
   RAW_Input.SB00_0 := TRUE;
   RAW_Input.SB00_6 := TRUE;
   RAW_Input.SB01 := 16#02;
   RAW_Input.SW02 := 16#1194;
   RAW_Input.SW04 := 292;
   RAW_Input.SW08 := 629;
   RAW_Input.SW22 := 16#FED3;
   RAW_Output.CB01 := 16#01;
   RAW_Output.CW02 := 16#1194;
   RAW_Output.CW08 := 16#0001;
   IHK.DelSTR_Timer_PV := 1;
   IHK.DelSTP_Timer_PV := 3;
   IHK.DelSTP_Timer_Mem := 3;
   IHK.RES_Timer_PV := 2;
   IHK.RES_Timer_Mem := 2;
   IHK.ChgOverTime_PV := 1;
   IHK.ChgOverTime_Mem := 1;
   IHK.CoastTimer_PV := 1;
   IHK.CoastTimer_Mem := 1;
   IHK.DelSTR_Timer_DN := TRUE;
   IHK.AUX_DelSTR_Time := 1;
   IHK.CoastSTP := TRUE;
   IHK.ComON := TRUE;
   IHK.Aux_CB01_0 := TRUE;
   IHK.No_Acyc := TRUE;
   IHK.Pulse._01 := TRUE;
   IHK.Pulse._03 := TRUE;
   AC.Ons_Read_Req := TRUE;
   AC.Motor_Data_99._06 := 100.0;
   AC.Motor_Data_99._09 := 100;
   AC.Motor_Data_99._10 := 100.0;
   AC._99_Status := 16#0000_0000;
   AC_Read_99_Migra.STATUS := 16#0000_0000;
   OUT.MCC := TRUE;
   OUT.RDY := TRUE;
   OUT.OVL := TRUE;
   OUT.RET1 := TRUE;
   OUT.LSTP := TRUE;
   OUT.REM := TRUE;
   OUT.SSW := TRUE;
   OUT.TFA := TRUE;
   OUT.DRDY := TRUE;
   OUT.STALL := TRUE;
   OUT.EARTH := TRUE;
   OUT.UBAL := TRUE;
   OUT.GFA := TRUE;
   OUT.GWA := TRUE;
   OUT.BUSF := TRUE;
   OUT.DOPR := TRUE;
   OUT.AI1 := 62.9;
   OUT.AI2 := 29.2;
   OUT.AI3 := 90.0;
END_DATA_BLOCK

DATA_BLOCK "_2010CV120M01_AD"   // DB14009
TITLE = Instance DB Adapter Block: _1010CV120M01
{ S7_Optimized_Access := 'FALSE' }
AUTHOR : 7Art
NAME : APPT_DB
VERSION : 8.0
// stored: InstanceOfName IUSYS_3UF70_V5_MOTOR
"IUSYS_3UF70_V5_MOTOR"
BEGIN
   INREF := 570;
   OUTREF := 570;
   FUNCTYPE := 41;
   NET := 101;
   NODE := 25;
   MCC := TRUE;
   RDY := TRUE;
   OVL := TRUE;
   RET1 := TRUE;
   LSTR1 := TRUE;
   REM := TRUE;
   SSW := TRUE;
   TFA := TRUE;
   DRDY := TRUE;
   STALL := TRUE;
   EARTH := TRUE;
   UBAL := TRUE;
   GFA := TRUE;
   GWA := TRUE;
   BUSF := TRUE;
   DOPR := TRUE;
   ES := TRUE;
   AI1 := 25.0;
   Raw_InPut.SB00_0 := TRUE;
   Raw_InPut.SB00_2 := TRUE;
   Raw_InPut.SB00_3 := TRUE;
   Raw_InPut.SB00_4 := TRUE;
   Raw_InPut.SB01_3 := TRUE;
   Raw_InPut.SW02 := 25;
   Raw_OutPut.CB00_0 := TRUE;
   Raw_OutPut.CB00_3 := TRUE;
   Raw_OutPut.CB00_7 := TRUE;
   IHK.Ret1_old := TRUE;
   OUT.MCC := TRUE;
   OUT.RDY := TRUE;
   OUT.OVL := TRUE;
   OUT.RET1 := TRUE;
   OUT.LSTR1 := TRUE;
   OUT.REM := TRUE;
   OUT.SSW := TRUE;
   OUT.TFA := TRUE;
   OUT.DRDY := TRUE;
   OUT.STALL := TRUE;
   OUT.EARTH := TRUE;
   OUT.UBAL := TRUE;
   OUT.GFA := TRUE;
   OUT.GWA := TRUE;
   OUT.BUSF := TRUE;
   OUT.DOPR := TRUE;
   OUT.ES := TRUE;
   OUT.AI1 := 25.0;
END_DATA_BLOCK

DATA_BLOCK "_2010BF110U01_AD"   // DB14011
{ S7_Optimized_Access := 'FALSE' }
VERSION : 0.1
// stored: InstanceOfName IUSYS_ALTIVAR_MB_MOTOR
"IUSYS_ALTIVAR_MB_MOTOR"
BEGIN
   CV := 30.0;
   Frame1_PTR_0 := 1591;
   Frame1_PTR_2 := 150;
   Frame1_PTR_3 := 1221;
   Frame1_PTR_6 := 4035;
   Frame2_PTR_0 := 500;
   MCC := TRUE;
   RDY := TRUE;
   OVL := TRUE;
   RET1 := TRUE;
   LSTP := TRUE;
   REM := TRUE;
   SSW := TRUE;
   TFA := TRUE;
   DRDY := TRUE;
   STALL := TRUE;
   EARTH := TRUE;
   UBAL := TRUE;
   GFA := TRUE;
   GWA := TRUE;
   BUSF := TRUE;
   DOPR := TRUE;
   AI1 := 122.1;
   AI2 := 403.5;
   AI3 := 30.0;
   Frame5_PTR_0 := 1;
   Frame5_PTR_1 := 150;
   IHK.RES_Timer_PV := 2;
   IHK.RES_Timer_Mem := 2;
   IHK.Aux_CB01_0 := TRUE;
   AC._99_Status := 16#0000_0000;
   AC_Read_99_Migra.STATUS := 16#0000_0000;
   OUT.MCC := TRUE;
   OUT.RDY := TRUE;
   OUT.OVL := TRUE;
   OUT.RET1 := TRUE;
   OUT.LSTP := TRUE;
   OUT.REM := TRUE;
   OUT.SSW := TRUE;
   OUT.TFA := TRUE;
   OUT.DRDY := TRUE;
   OUT.STALL := TRUE;
   OUT.EARTH := TRUE;
   OUT.UBAL := TRUE;
   OUT.GFA := TRUE;
   OUT.GWA := TRUE;
   OUT.BUSF := TRUE;
   OUT.DOPR := TRUE;
   OUT.AI1 := 122.1;
   OUT.AI2 := 403.5;
   OUT.AI3 := 30.0;
   cmd_old := 1;
   set_spd_old := 150;
END_DATA_BLOCK

DATA_BLOCK "_2010SC130U01_AD"   // DB14012
{ S7_Optimized_Access := 'FALSE' }
VERSION : 0.1
// stored: InstanceOfName IUSYS_ALTIVAR_MB_MOTOR
"IUSYS_ALTIVAR_MB_MOTOR"
BEGIN
   CV := 100.0;
   Frame1_PTR_0 := 1591;
   Frame1_PTR_2 := 500;
   Frame1_PTR_3 := 497;
   Frame1_PTR_6 := 4056;
   Frame2_PTR_0 := 500;
   MCC := TRUE;
   RDY := TRUE;
   OVL := TRUE;
   RET1 := TRUE;
   LSTP := TRUE;
   REM := TRUE;
   SSW := TRUE;
   TFA := TRUE;
   DRDY := TRUE;
   STALL := TRUE;
   EARTH := TRUE;
   UBAL := TRUE;
   GFA := TRUE;
   GWA := TRUE;
   BUSF := TRUE;
   DOPR := TRUE;
   AI1 := 49.7;
   AI2 := 405.6;
   AI3 := 100.0;
   Frame5_PTR_0 := 1;
   Frame5_PTR_1 := 500;
   IHK.RES_Timer_PV := 2;
   IHK.RES_Timer_Mem := 2;
   IHK.Aux_CB01_0 := TRUE;
   AC._99_Status := 16#0000_0000;
   AC_Read_99_Migra.STATUS := 16#0000_0000;
   OUT.MCC := TRUE;
   OUT.RDY := TRUE;
   OUT.OVL := TRUE;
   OUT.RET1 := TRUE;
   OUT.LSTP := TRUE;
   OUT.REM := TRUE;
   OUT.SSW := TRUE;
   OUT.TFA := TRUE;
   OUT.DRDY := TRUE;
   OUT.STALL := TRUE;
   OUT.EARTH := TRUE;
   OUT.UBAL := TRUE;
   OUT.GFA := TRUE;
   OUT.GWA := TRUE;
   OUT.BUSF := TRUE;
   OUT.DOPR := TRUE;
   OUT.AI1 := 49.7;
   OUT.AI2 := 405.6;
   OUT.AI3 := 100.0;
   cmd_old := 1;
   set_spd_old := 500;
END_DATA_BLOCK

DATA_BLOCK "_2010SJ950M01_AD"   // DB14110
TITLE = Instance DB Adapter Block: _2010SJ950M01
{ S7_Optimized_Access := 'FALSE' }
AUTHOR : METIS
NAME : APPT_DB
VERSION : 8.0
// stored: InstanceOfName IUSYS_3UF70_V5_MOTOR
"IUSYS_3UF70_V5_MOTOR"
BEGIN
   INREF := 5186;
   OUTREF := 5186;
   FUNCTYPE := 41;
   NET := 106;
   NODE := 26;
   MCC := TRUE;
   RDY := TRUE;
   OVL := TRUE;
   REM := TRUE;
   SSW := TRUE;
   TFA := TRUE;
   STALL := TRUE;
   EARTH := TRUE;
   UBAL := TRUE;
   GWA := TRUE;
   DTEST := TRUE;
   ES := TRUE;
   Raw_OutPut.CB00_2 := TRUE;
   Raw_OutPut.CB00_3 := TRUE;
   Raw_OutPut.CB00_7 := TRUE;
   OUT.MCC := TRUE;
   OUT.RDY := TRUE;
   OUT.OVL := TRUE;
   OUT.REM := TRUE;
   OUT.SSW := TRUE;
   OUT.TFA := TRUE;
   OUT.STALL := TRUE;
   OUT.EARTH := TRUE;
   OUT.UBAL := TRUE;
   OUT.GWA := TRUE;
   OUT.DTEST := TRUE;
   OUT.ES := TRUE;
END_DATA_BLOCK

